  PROC DrawPart253()
    MoveL Offs(pOrigin,224.94,44.31,6.00),vTravel,z5,tPen\WObj:=wPaper;
    MoveL Offs(pOrigin,224.94,44.31,0.00),v60,z0,tPen\WObj:=wPaper;
    MoveL Offs(pOrigin,224.94,40.70,0.00),v40,z0,tPen\WObj:=wPaper;
    MoveL Offs(pOrigin,224.78,39.89,0.00),v40,z0,tPen\WObj:=wPaper;
    MoveL Offs(pOrigin,227.34,42.45,0.00),v40,z0,tPen\WObj:=wPaper;
    MoveL Offs(pOrigin,226.84,42.46,0.00),v40,z0,tPen\WObj:=wPaper;
    MoveL Offs(pOrigin,223.22,42.46,0.00),v40,fine,tPen\WObj:=wPaper;
    MoveL Offs(pOrigin,223.22,42.46,6.00),v60,z5,tPen\WObj:=wPaper;
    MoveL Offs(pOrigin,222.09,40.18,6.00),vTravel,z5,tPen\WObj:=wPaper;
    MoveL Offs(pOrigin,222.09,40.18,0.00),v60,z0,tPen\WObj:=wPaper;
    MoveL Offs(pOrigin,226.29,44.39,0.00),v40,z0,tPen\WObj:=wPaper;
    MoveL Offs(pOrigin,226.74,43.34,0.00),v40,z0,tPen\WObj:=wPaper;
    MoveL Offs(pOrigin,223.28,39.89,0.00),v40,z0,tPen\WObj:=wPaper;
    MoveL Offs(pOrigin,223.66,39.43,0.00),v40,z0,tPen\WObj:=wPaper;
    MoveL Offs(pOrigin,205.18,57.91,0.00),v40,z0,tPen\WObj:=wPaper;
    MoveL Offs(pOrigin,204.91,57.36,0.00),v40,z0,tPen\WObj:=wPaper;
    MoveL Offs(pOrigin,203.56,56.00,0.00),v40,z0,tPen\WObj:=wPaper;
    MoveL Offs(pOrigin,203.09,55.52,0.00),v40,z0,tPen\WObj:=wPaper;
    MoveL Offs(pOrigin,197.53,61.08,0.00),v40,z0,tPen\WObj:=wPaper;
    MoveL Offs(pOrigin,197.58,60.48,0.00),v40,z0,tPen\WObj:=wPaper;
    MoveL Offs(pOrigin,196.23,59.13,0.00),v40,z0,tPen\WObj:=wPaper;
    MoveL Offs(pOrigin,196.66,59.35,0.00),v40,z0,tPen\WObj:=wPaper;
    MoveL Offs(pOrigin,199.00,59.35,0.00),v40,z0,tPen\WObj:=wPaper;
    MoveL Offs(pOrigin,198.78,60.18,0.00),v40,z0,tPen\WObj:=wPaper;
    MoveL Offs(pOrigin,197.28,58.68,0.00),v40,z0,tPen\WObj:=wPaper;
    MoveL Offs(pOrigin,197.69,57.93,0.00),v40,z0,tPen\WObj:=wPaper;
    MoveL Offs(pOrigin,193.48,62.14,0.00),v40,z0,tPen\WObj:=wPaper;
    MoveL Offs(pOrigin,192.94,61.81,0.00),v40,z0,tPen\WObj:=wPaper;
    MoveL Offs(pOrigin,191.74,60.61,0.00),v40,z0,tPen\WObj:=wPaper;
    MoveL Offs(pOrigin,191.39,59.75,0.00),v40,z0,tPen\WObj:=wPaper;
    MoveL Offs(pOrigin,187.04,64.10,0.00),v40,z0,tPen\WObj:=wPaper;
    MoveL Offs(pOrigin,186.95,63.29,0.00),v40,z0,tPen\WObj:=wPaper;
    MoveL Offs(pOrigin,186.05,62.39,0.00),v40,z0,tPen\WObj:=wPaper;
    MoveL Offs(pOrigin,187.10,61.95,0.00),v40,z0,tPen\WObj:=wPaper;
    MoveL Offs(pOrigin,188.30,63.15,0.00),v40,z0,tPen\WObj:=wPaper;
    MoveL Offs(pOrigin,189.44,63.20,0.00),v40,z0,tPen\WObj:=wPaper;
    MoveL Offs(pOrigin,193.49,59.14,0.00),v40,z0,tPen\WObj:=wPaper;
    MoveL Offs(pOrigin,193.98,59.87,0.00),v40,z0,tPen\WObj:=wPaper;
    MoveL Offs(pOrigin,195.34,61.22,0.00),v40,z0,tPen\WObj:=wPaper;
    MoveL Offs(pOrigin,195.43,61.68,0.00),v40,z0,tPen\WObj:=wPaper;
    MoveL Offs(pOrigin,200.39,56.72,0.00),v40,z0,tPen\WObj:=wPaper;
    MoveL Offs(pOrigin,200.72,57.64,0.00),v40,z0,tPen\WObj:=wPaper;
    MoveL Offs(pOrigin,202.07,59.00,0.00),v40,z0,tPen\WObj:=wPaper;
    MoveL Offs(pOrigin,202.48,59.11,0.00),v40,z0,tPen\WObj:=wPaper;
    MoveL Offs(pOrigin,210.15,51.45,0.00),v40,z0,tPen\WObj:=wPaper;
    MoveL Offs(pOrigin,210.14,52.13,0.00),v40,z0,tPen\WObj:=wPaper;
    MoveL Offs(pOrigin,211.79,53.78,0.00),v40,z0,tPen\WObj:=wPaper;
    MoveL Offs(pOrigin,211.33,54.74,0.00),v40,z0,tPen\WObj:=wPaper;
    MoveL Offs(pOrigin,226.96,39.12,0.00),v40,z0,tPen\WObj:=wPaper;
    MoveL Offs(pOrigin,227.63,39.75,0.00),v40,z0,tPen\WObj:=wPaper;
    MoveL Offs(pOrigin,229.58,41.70,0.00),v40,fine,tPen\WObj:=wPaper;
    MoveL Offs(pOrigin,229.58,41.70,6.00),v60,z5,tPen\WObj:=wPaper;
    MoveL Offs(pOrigin,227.05,41.55,6.00),vTravel,z5,tPen\WObj:=wPaper;
    MoveL Offs(pOrigin,227.05,41.55,0.00),v60,z0,tPen\WObj:=wPaper;
    MoveL Offs(pOrigin,227.05,40.49,0.00),v40,fine,tPen\WObj:=wPaper;
    MoveL Offs(pOrigin,227.05,40.49,6.00),v60,z5,tPen\WObj:=wPaper;
    MoveL Offs(pOrigin,225.46,39.12,6.00),vTravel,z5,tPen\WObj:=wPaper;
    MoveL Offs(pOrigin,225.46,39.12,0.00),v60,z0,tPen\WObj:=wPaper;
    MoveL Offs(pOrigin,208.78,55.80,0.00),v40,z0,tPen\WObj:=wPaper;
    MoveL Offs(pOrigin,208.80,55.27,0.00),v40,z0,tPen\WObj:=wPaper;
    MoveL Offs(pOrigin,207.45,53.92,0.00),v40,z0,tPen\WObj:=wPaper;
    MoveL Offs(pOrigin,207.92,54.07,0.00),v40,z0,tPen\WObj:=wPaper;
    MoveL Offs(pOrigin,209.84,54.07,0.00),v40,z0,tPen\WObj:=wPaper;
    MoveL Offs(pOrigin,209.85,54.83,0.00),v40,z0,tPen\WObj:=wPaper;
    MoveL Offs(pOrigin,208.34,53.32,0.00),v40,z0,tPen\WObj:=wPaper;
    MoveL Offs(pOrigin,209.39,52.88,0.00),v40,z0,tPen\WObj:=wPaper;
    MoveL Offs(pOrigin,210.74,54.23,0.00),v40,fine,tPen\WObj:=wPaper;
    MoveL Offs(pOrigin,210.74,54.23,6.00),v60,z5,tPen\WObj:=wPaper;
    MoveL Offs(pOrigin,209.62,53.02,6.00),vTravel,z5,tPen\WObj:=wPaper;
    MoveL Offs(pOrigin,209.62,53.02,0.00),v60,z0,tPen\WObj:=wPaper;
    MoveL Offs(pOrigin,218.76,53.02,0.00),v40,z0,tPen\WObj:=wPaper;
    MoveL Offs(pOrigin,218.98,52.81,0.00),v40,z0,tPen\WObj:=wPaper;
    MoveL Offs(pOrigin,217.91,53.88,0.00),v40,z0,tPen\WObj:=wPaper;
    MoveL Offs(pOrigin,218.98,52.81,0.00),v40,z0,tPen\WObj:=wPaper;
    MoveL Offs(pOrigin,218.98,53.51,0.00),v40,z0,tPen\WObj:=wPaper;
    MoveL Offs(pOrigin,217.03,51.55,0.00),v40,fine,tPen\WObj:=wPaper;
    MoveL Offs(pOrigin,217.03,51.55,6.00),v60,z5,tPen\WObj:=wPaper;
    MoveL Offs(pOrigin,215.79,53.88,6.00),vTravel,z5,tPen\WObj:=wPaper;
    MoveL Offs(pOrigin,215.79,53.88,0.00),v60,z0,tPen\WObj:=wPaper;
    MoveL Offs(pOrigin,216.21,54.30,0.00),v40,z0,tPen\WObj:=wPaper;
    MoveL Offs(pOrigin,215.79,53.88,0.00),v40,fine,tPen\WObj:=wPaper;
    MoveL Offs(pOrigin,215.79,53.88,6.00),v60,z5,tPen\WObj:=wPaper;
    MoveL Offs(pOrigin,216.64,55.13,6.00),vTravel,z5,tPen\WObj:=wPaper;
    MoveL Offs(pOrigin,216.64,55.13,0.00),v60,z0,tPen\WObj:=wPaper;
    MoveL Offs(pOrigin,217.91,55.13,0.00),v40,z0,tPen\WObj:=wPaper;
    MoveL Offs(pOrigin,217.91,56.18,0.00),v40,z0,tPen\WObj:=wPaper;
    MoveL Offs(pOrigin,216.85,56.18,0.00),v40,fine,tPen\WObj:=wPaper;
    MoveL Offs(pOrigin,216.85,56.18,6.00),v60,z5,tPen\WObj:=wPaper;
    MoveL Offs(pOrigin,218.66,57.87,6.00),vTravel,z5,tPen\WObj:=wPaper;
    MoveL Offs(pOrigin,218.66,57.87,0.00),v60,z0,tPen\WObj:=wPaper;
    MoveL Offs(pOrigin,208.75,67.78,0.00),v40,z0,tPen\WObj:=wPaper;
    MoveL Offs(pOrigin,208.84,67.26,0.00),v40,z0,tPen\WObj:=wPaper;
    MoveL Offs(pOrigin,207.33,65.75,0.00),v40,z0,tPen\WObj:=wPaper;
    MoveL Offs(pOrigin,206.36,65.69,0.00),v40,z0,tPen\WObj:=wPaper;
    MoveL Offs(pOrigin,192.23,79.82,0.00),v40,z0,tPen\WObj:=wPaper;
    MoveL Offs(pOrigin,192.24,79.04,0.00),v40,z0,tPen\WObj:=wPaper;
    MoveL Offs(pOrigin,188.19,74.98,0.00),v40,z0,tPen\WObj:=wPaper;
    MoveL Offs(pOrigin,188.16,75.19,0.00),v40,z0,tPen\WObj:=wPaper;
    MoveL Offs(pOrigin,206.65,75.19,0.00),v40,z0,tPen\WObj:=wPaper;
    MoveL Offs(pOrigin,206.86,74.14,0.00),v40,z0,tPen\WObj:=wPaper;
    MoveL Offs(pOrigin,210.48,74.14,0.00),v40,z0,tPen\WObj:=wPaper;
    MoveL Offs(pOrigin,210.51,74.90,0.00),v40,z0,tPen\WObj:=wPaper;
    MoveL Offs(pOrigin,208.85,73.25,0.00),v40,z0,tPen\WObj:=wPaper;
    MoveL Offs(pOrigin,208.58,72.43,0.00),v40,z0,tPen\WObj:=wPaper;
    MoveL Offs(pOrigin,204.53,76.48,0.00),v40,z0,tPen\WObj:=wPaper;
    MoveL Offs(pOrigin,204.52,76.38,0.00),v40,z0,tPen\WObj:=wPaper;
    MoveL Offs(pOrigin,202.72,74.58,0.00),v40,z0,tPen\WObj:=wPaper;
    MoveL Offs(pOrigin,202.74,73.79,0.00),v40,z0,tPen\WObj:=wPaper;
    MoveL Offs(pOrigin,199.58,76.95,0.00),v40,z0,tPen\WObj:=wPaper;
    MoveL Offs(pOrigin,200.18,76.52,0.00),v40,z0,tPen\WObj:=wPaper;
    MoveL Offs(pOrigin,195.37,71.71,0.00),v40,z0,tPen\WObj:=wPaper;
    MoveL Offs(pOrigin,195.60,72.02,0.00),v40,z0,tPen\WObj:=wPaper;
    MoveL Offs(pOrigin,199.00,72.02,0.00),v40,z0,tPen\WObj:=wPaper;
    MoveL Offs(pOrigin,199.21,72.36,0.00),v40,z0,tPen\WObj:=wPaper;
    MoveL Offs(pOrigin,199.43,71.94,0.00),v40,z0,tPen\WObj:=wPaper;
    MoveL Offs(pOrigin,199.21,72.36,0.00),v40,z0,tPen\WObj:=wPaper;
    MoveL Offs(pOrigin,199.42,72.77,0.00),v40,z0,tPen\WObj:=wPaper;
    MoveL Offs(pOrigin,197.61,70.97,0.00),v40,z0,tPen\WObj:=wPaper;
    MoveL Offs(pOrigin,197.94,70.97,0.00),v40,z0,tPen\WObj:=wPaper;
    MoveL Offs(pOrigin,200.49,70.97,0.00),v40,z0,tPen\WObj:=wPaper;
  ENDPROC

  PROC DrawPart254()
    MoveL Offs(pOrigin,201.06,71.43,0.00),v40,z0,tPen\WObj:=wPaper;
    MoveL Offs(pOrigin,199.71,70.07,0.00),v40,z0,tPen\WObj:=wPaper;
    MoveL Offs(pOrigin,199.90,69.16,0.00),v40,z0,tPen\WObj:=wPaper;
    MoveL Offs(pOrigin,171.05,98.01,0.00),v40,z0,tPen\WObj:=wPaper;
    MoveL Offs(pOrigin,170.58,97.70,0.00),v40,z0,tPen\WObj:=wPaper;
    MoveL Offs(pOrigin,165.32,92.44,0.00),v40,z0,tPen\WObj:=wPaper;
    MoveL Offs(pOrigin,165.64,92.55,0.00),v40,z0,tPen\WObj:=wPaper;
    MoveL Offs(pOrigin,165.21,93.19,0.00),v40,z0,tPen\WObj:=wPaper;
    MoveL Offs(pOrigin,165.64,92.55,0.00),v40,z0,tPen\WObj:=wPaper;
    MoveL Offs(pOrigin,165.42,93.14,0.00),v40,z0,tPen\WObj:=wPaper;
    MoveL Offs(pOrigin,167.98,93.14,0.00),v40,z0,tPen\WObj:=wPaper;
    MoveL Offs(pOrigin,167.98,93.40,0.00),v40,z0,tPen\WObj:=wPaper;
    MoveL Offs(pOrigin,168.12,92.34,0.00),v40,z0,tPen\WObj:=wPaper;
    MoveL Offs(pOrigin,168.82,91.28,0.00),v40,z0,tPen\WObj:=wPaper;
    MoveL Offs(pOrigin,170.31,90.85,0.00),v40,z0,tPen\WObj:=wPaper;
    MoveL Offs(pOrigin,170.52,89.98,0.00),v40,z0,tPen\WObj:=wPaper;
    MoveL Offs(pOrigin,168.19,89.98,0.00),v40,z0,tPen\WObj:=wPaper;
    MoveL Offs(pOrigin,167.76,90.00,0.00),v40,z0,tPen\WObj:=wPaper;
    MoveL Offs(pOrigin,167.12,90.64,0.00),v40,z0,tPen\WObj:=wPaper;
    MoveL Offs(pOrigin,167.76,90.00,0.00),v40,z0,tPen\WObj:=wPaper;
    MoveL Offs(pOrigin,167.41,90.05,0.00),v40,z0,tPen\WObj:=wPaper;
    MoveL Offs(pOrigin,170.27,92.90,0.00),v40,z0,tPen\WObj:=wPaper;
    MoveL Offs(pOrigin,171.02,93.65,0.00),v40,z0,tPen\WObj:=wPaper;
    MoveL Offs(pOrigin,173.87,96.51,0.00),v40,z0,tPen\WObj:=wPaper;
    MoveL Offs(pOrigin,172.98,97.11,0.00),v40,z0,tPen\WObj:=wPaper;
    MoveL Offs(pOrigin,170.42,94.55,0.00),v40,z0,tPen\WObj:=wPaper;
    MoveL Offs(pOrigin,169.68,95.26,0.00),v40,z0,tPen\WObj:=wPaper;
    MoveL Offs(pOrigin,173.92,95.26,0.00),v40,z0,tPen\WObj:=wPaper;
    MoveL Offs(pOrigin,174.47,95.61,0.00),v40,z0,tPen\WObj:=wPaper;
    MoveL Offs(pOrigin,171.92,93.06,0.00),v40,z0,tPen\WObj:=wPaper;
    MoveL Offs(pOrigin,172.66,92.31,0.00),v40,z0,tPen\WObj:=wPaper;
    MoveL Offs(pOrigin,175.22,94.87,0.00),v40,z0,tPen\WObj:=wPaper;
    MoveL Offs(pOrigin,174.99,94.46,0.00),v40,z0,tPen\WObj:=wPaper;
    MoveL Offs(pOrigin,174.35,95.10,0.00),v40,z0,tPen\WObj:=wPaper;
    MoveL Offs(pOrigin,174.99,94.46,0.00),v40,z0,tPen\WObj:=wPaper;
    MoveL Offs(pOrigin,175.20,94.20,0.00),v40,z0,tPen\WObj:=wPaper;
    MoveL Offs(pOrigin,172.01,94.20,0.00),v40,fine,tPen\WObj:=wPaper;
    MoveL Offs(pOrigin,172.01,94.20,6.00),v60,z5,tPen\WObj:=wPaper;
    MoveL Offs(pOrigin,173.08,93.14,6.00),vTravel,z5,tPen\WObj:=wPaper;
    MoveL Offs(pOrigin,173.08,93.14,0.00),v60,z0,tPen\WObj:=wPaper;
    MoveL Offs(pOrigin,176.69,93.14,0.00),v40,z0,tPen\WObj:=wPaper;
    MoveL Offs(pOrigin,176.90,92.97,0.00),v40,z0,tPen\WObj:=wPaper;
    MoveL Offs(pOrigin,176.48,93.40,0.00),v40,z0,tPen\WObj:=wPaper;
    MoveL Offs(pOrigin,176.90,92.97,0.00),v40,z0,tPen\WObj:=wPaper;
    MoveL Offs(pOrigin,176.86,93.52,0.00),v40,z0,tPen\WObj:=wPaper;
    MoveL Offs(pOrigin,174.31,90.97,0.00),v40,z0,tPen\WObj:=wPaper;
    MoveL Offs(pOrigin,173.56,91.71,0.00),v40,z0,tPen\WObj:=wPaper;
    MoveL Offs(pOrigin,175.96,94.12,0.00),v40,z0,tPen\WObj:=wPaper;
    MoveL Offs(pOrigin,176.05,93.61,0.00),v40,z0,tPen\WObj:=wPaper;
    MoveL Offs(pOrigin,175.41,94.25,0.00),v40,z0,tPen\WObj:=wPaper;
    MoveL Offs(pOrigin,176.05,93.61,0.00),v40,fine,tPen\WObj:=wPaper;
    MoveL Offs(pOrigin,176.05,93.61,6.00),v60,z5,tPen\WObj:=wPaper;
    MoveL Offs(pOrigin,174.35,92.09,6.00),vTravel,z5,tPen\WObj:=wPaper;
    MoveL Offs(pOrigin,174.35,92.09,0.00),v60,z0,tPen\WObj:=wPaper;
    MoveL Offs(pOrigin,177.96,92.09,0.00),v40,z0,tPen\WObj:=wPaper;
    MoveL Offs(pOrigin,178.65,92.33,0.00),v40,z0,tPen\WObj:=wPaper;
    MoveL Offs(pOrigin,175.95,89.62,0.00),v40,z0,tPen\WObj:=wPaper;
    MoveL Offs(pOrigin,176.90,89.98,0.00),v40,z0,tPen\WObj:=wPaper;
    MoveL Offs(pOrigin,180.30,89.98,0.00),v40,z0,tPen\WObj:=wPaper;
    MoveL Offs(pOrigin,181.04,90.24,0.00),v40,z0,tPen\WObj:=wPaper;
    MoveL Offs(pOrigin,178.49,87.69,0.00),v40,z0,tPen\WObj:=wPaper;
    MoveL Offs(pOrigin,179.45,87.86,0.00),v40,z0,tPen\WObj:=wPaper;
    MoveL Offs(pOrigin,182.85,87.86,0.00),v40,z0,tPen\WObj:=wPaper;
    MoveL Offs(pOrigin,183.28,88.00,0.00),v40,z0,tPen\WObj:=wPaper;
    MoveL Offs(pOrigin,180.73,85.44,0.00),v40,z0,tPen\WObj:=wPaper;
    MoveL Offs(pOrigin,181.63,84.85,0.00),v40,z0,tPen\WObj:=wPaper;
    MoveL Offs(pOrigin,184.18,87.40,0.00),v40,z0,tPen\WObj:=wPaper;
    MoveL Offs(pOrigin,183.70,87.24,0.00),v40,z0,tPen\WObj:=wPaper;
    MoveL Offs(pOrigin,182.85,88.09,0.00),v40,z0,tPen\WObj:=wPaper;
    MoveL Offs(pOrigin,183.70,87.24,0.00),v40,z0,tPen\WObj:=wPaper;
    MoveL Offs(pOrigin,184.12,86.81,0.00),v40,z0,tPen\WObj:=wPaper;
    MoveL Offs(pOrigin,180.94,86.81,0.00),v40,z0,tPen\WObj:=wPaper;
    MoveL Offs(pOrigin,180.13,86.34,0.00),v40,z0,tPen\WObj:=wPaper;
    MoveL Offs(pOrigin,182.54,88.75,0.00),v40,z0,tPen\WObj:=wPaper;
    MoveL Offs(pOrigin,182.00,88.72,0.00),v40,z0,tPen\WObj:=wPaper;
    MoveL Offs(pOrigin,181.15,89.57,0.00),v40,z0,tPen\WObj:=wPaper;
    MoveL Offs(pOrigin,182.00,88.72,0.00),v40,z0,tPen\WObj:=wPaper;
    MoveL Offs(pOrigin,181.58,88.92,0.00),v40,z0,tPen\WObj:=wPaper;
    MoveL Offs(pOrigin,178.18,88.92,0.00),v40,fine,tPen\WObj:=wPaper;
    MoveL Offs(pOrigin,178.18,88.92,6.00),v60,z5,tPen\WObj:=wPaper;
    MoveL Offs(pOrigin,176.70,88.88,6.00),vTravel,z5,tPen\WObj:=wPaper;
    MoveL Offs(pOrigin,176.70,88.88,0.00),v60,z0,tPen\WObj:=wPaper;
    MoveL Offs(pOrigin,179.40,91.58,0.00),v40,fine,tPen\WObj:=wPaper;
    MoveL Offs(pOrigin,179.40,91.58,6.00),v60,z5,tPen\WObj:=wPaper;
    MoveL Offs(pOrigin,181.64,89.34,6.00),vTravel,z5,tPen\WObj:=wPaper;
    MoveL Offs(pOrigin,181.64,89.34,0.00),v60,z0,tPen\WObj:=wPaper;
    MoveL Offs(pOrigin,179.24,86.94,0.00),v40,fine,tPen\WObj:=wPaper;
    MoveL Offs(pOrigin,179.24,86.94,6.00),v60,z5,tPen\WObj:=wPaper;
    MoveL Offs(pOrigin,182.00,85.75,6.00),vTravel,z5,tPen\WObj:=wPaper;
    MoveL Offs(pOrigin,182.00,85.75,0.00),v60,z0,tPen\WObj:=wPaper;
    MoveL Offs(pOrigin,184.98,85.75,0.00),v40,z0,tPen\WObj:=wPaper;
    MoveL Offs(pOrigin,185.40,85.75,0.00),v40,z0,tPen\WObj:=wPaper;
    MoveL Offs(pOrigin,184.34,86.81,0.00),v40,z0,tPen\WObj:=wPaper;
    MoveL Offs(pOrigin,185.40,85.75,0.00),v40,z0,tPen\WObj:=wPaper;
    MoveL Offs(pOrigin,185.83,86.06,0.00),v40,z0,tPen\WObj:=wPaper;
    MoveL Offs(pOrigin,183.12,83.36,0.00),v40,z0,tPen\WObj:=wPaper;
    MoveL Offs(pOrigin,182.37,84.10,0.00),v40,z0,tPen\WObj:=wPaper;
    MoveL Offs(pOrigin,184.93,86.66,0.00),v40,fine,tPen\WObj:=wPaper;
    MoveL Offs(pOrigin,184.93,86.66,6.00),v60,z5,tPen\WObj:=wPaper;
    MoveL Offs(pOrigin,183.37,88.68,6.00),vTravel,z5,tPen\WObj:=wPaper;
    MoveL Offs(pOrigin,183.37,88.68,0.00),v60,z0,tPen\WObj:=wPaper;
    MoveL Offs(pOrigin,191.33,80.72,0.00),v40,z0,tPen\WObj:=wPaper;
    MoveL Offs(pOrigin,190.75,80.53,0.00),v40,z0,tPen\WObj:=wPaper;
    MoveL Offs(pOrigin,185.94,75.72,0.00),v40,z0,tPen\WObj:=wPaper;
    MoveL Offs(pOrigin,185.19,76.25,0.00),v40,z0,tPen\WObj:=wPaper;
    MoveL Offs(pOrigin,189.23,76.25,0.00),v40,fine,tPen\WObj:=wPaper;
    MoveL Offs(pOrigin,189.23,76.25,6.00),v60,z5,tPen\WObj:=wPaper;
    MoveL Offs(pOrigin,190.50,77.30,6.00),vTravel,z5,tPen\WObj:=wPaper;
    MoveL Offs(pOrigin,190.50,77.30,0.00),v60,z0,tPen\WObj:=wPaper;
    MoveL Offs(pOrigin,193.48,77.30,0.00),v40,z0,tPen\WObj:=wPaper;
    MoveL Offs(pOrigin,193.89,77.70,0.00),v40,z0,tPen\WObj:=wPaper;
    MoveL Offs(pOrigin,190.28,74.09,0.00),v40,z0,tPen\WObj:=wPaper;
    MoveL Offs(pOrigin,190.92,74.14,0.00),v40,z0,tPen\WObj:=wPaper;
    MoveL Offs(pOrigin,197.30,74.14,0.00),v40,z0,tPen\WObj:=wPaper;
    MoveL Offs(pOrigin,197.51,73.85,0.00),v40,z0,tPen\WObj:=wPaper;
    MoveL Offs(pOrigin,197.73,73.43,0.00),v40,z0,tPen\WObj:=wPaper;
    MoveL Offs(pOrigin,197.51,73.85,0.00),v40,z0,tPen\WObj:=wPaper;
    MoveL Offs(pOrigin,197.49,73.21,0.00),v40,z0,tPen\WObj:=wPaper;
    MoveL Offs(pOrigin,197.49,71.72,0.00),v40,z0,tPen\WObj:=wPaper;
    MoveL Offs(pOrigin,196.57,71.41,0.00),v40,z0,tPen\WObj:=wPaper;
  ENDPROC

  PROC DrawPart255()
    MoveL Offs(pOrigin,198.52,73.37,0.00),v40,z0,tPen\WObj:=wPaper;
    MoveL Offs(pOrigin,198.15,73.21,0.00),v40,z0,tPen\WObj:=wPaper;
    MoveL Offs(pOrigin,198.57,73.00,0.00),v40,z0,tPen\WObj:=wPaper;
    MoveL Offs(pOrigin,198.15,73.21,0.00),v40,z0,tPen\WObj:=wPaper;
    MoveL Offs(pOrigin,198.15,73.08,0.00),v40,z0,tPen\WObj:=wPaper;
    MoveL Offs(pOrigin,193.26,73.08,0.00),v40,z0,tPen\WObj:=wPaper;
    MoveL Offs(pOrigin,193.57,72.90,0.00),v40,z0,tPen\WObj:=wPaper;
    MoveL Offs(pOrigin,197.33,76.66,0.00),v40,z0,tPen\WObj:=wPaper;
    MoveL Offs(pOrigin,198.08,76.95,0.00),v40,z0,tPen\WObj:=wPaper;
    MoveL Offs(pOrigin,201.09,73.95,0.00),v40,z0,tPen\WObj:=wPaper;
    MoveL Offs(pOrigin,201.22,74.57,0.00),v40,z0,tPen\WObj:=wPaper;
    MoveL Offs(pOrigin,203.02,76.38,0.00),v40,z0,tPen\WObj:=wPaper;
    MoveL Offs(pOrigin,202.73,76.79,0.00),v40,z0,tPen\WObj:=wPaper;
    MoveL Offs(pOrigin,206.48,73.03,0.00),v40,z0,tPen\WObj:=wPaper;
    MoveL Offs(pOrigin,206.61,73.99,0.00),v40,z0,tPen\WObj:=wPaper;
    MoveL Offs(pOrigin,208.26,75.64,0.00),v40,fine,tPen\WObj:=wPaper;
    MoveL Offs(pOrigin,208.26,75.64,6.00),v60,z5,tPen\WObj:=wPaper;
    MoveL Offs(pOrigin,209.46,75.35,6.00),vTravel,z5,tPen\WObj:=wPaper;
    MoveL Offs(pOrigin,209.46,75.35,0.00),v60,z0,tPen\WObj:=wPaper;
    MoveL Offs(pOrigin,207.66,73.54,0.00),v40,fine,tPen\WObj:=wPaper;
    MoveL Offs(pOrigin,207.66,73.54,6.00),v60,z5,tPen\WObj:=wPaper;
    MoveL Offs(pOrigin,210.05,72.95,6.00),vTravel,z5,tPen\WObj:=wPaper;
    MoveL Offs(pOrigin,210.05,72.95,0.00),v60,z0,tPen\WObj:=wPaper;
    MoveL Offs(pOrigin,211.55,74.45,0.00),v40,fine,tPen\WObj:=wPaper;
    MoveL Offs(pOrigin,211.55,74.45,6.00),v60,z5,tPen\WObj:=wPaper;
    MoveL Offs(pOrigin,210.22,75.27,6.00),vTravel,z5,tPen\WObj:=wPaper;
    MoveL Offs(pOrigin,210.22,75.27,0.00),v60,z0,tPen\WObj:=wPaper;
    MoveL Offs(pOrigin,218.64,66.85,0.00),v40,fine,tPen\WObj:=wPaper;
    MoveL Offs(pOrigin,218.64,66.85,6.00),v60,z5,tPen\WObj:=wPaper;
    MoveL Offs(pOrigin,218.50,64.01,6.00),vTravel,z5,tPen\WObj:=wPaper;
    MoveL Offs(pOrigin,218.50,64.01,0.00),v60,z0,tPen\WObj:=wPaper;
    MoveL Offs(pOrigin,212.64,69.87,0.00),v40,z0,tPen\WObj:=wPaper;
    MoveL Offs(pOrigin,213.34,70.27,0.00),v40,z0,tPen\WObj:=wPaper;
    MoveL Offs(pOrigin,214.99,71.92,0.00),v40,z0,tPen\WObj:=wPaper;
    MoveL Offs(pOrigin,214.94,71.09,0.00),v40,z0,tPen\WObj:=wPaper;
    MoveL Offs(pOrigin,214.73,71.51,0.00),v40,z0,tPen\WObj:=wPaper;
    MoveL Offs(pOrigin,214.94,71.09,0.00),v40,z0,tPen\WObj:=wPaper;
    MoveL Offs(pOrigin,214.94,70.97,0.00),v40,z0,tPen\WObj:=wPaper;
    MoveL Offs(pOrigin,213.45,70.97,0.00),v40,z0,tPen\WObj:=wPaper;
    MoveL Offs(pOrigin,213.88,70.03,0.00),v40,z0,tPen\WObj:=wPaper;
    MoveL Offs(pOrigin,213.66,70.45,0.00),v40,z0,tPen\WObj:=wPaper;
    MoveL Offs(pOrigin,213.88,70.03,0.00),v40,fine,tPen\WObj:=wPaper;
    MoveL Offs(pOrigin,213.88,70.03,6.00),v60,z5,tPen\WObj:=wPaper;
    MoveL Offs(pOrigin,214.09,72.02,6.00),vTravel,z5,tPen\WObj:=wPaper;
    MoveL Offs(pOrigin,214.09,72.02,0.00),v60,z0,tPen\WObj:=wPaper;
    MoveL Offs(pOrigin,212.18,72.02,0.00),v40,z0,tPen\WObj:=wPaper;
    MoveL Offs(pOrigin,211.96,72.15,0.00),v40,z0,tPen\WObj:=wPaper;
    MoveL Offs(pOrigin,212.46,71.80,0.00),v40,z0,tPen\WObj:=wPaper;
    MoveL Offs(pOrigin,210.26,73.07,0.00),v40,z0,tPen\WObj:=wPaper;
    MoveL Offs(pOrigin,205.16,74.49,0.00),v40,z0,tPen\WObj:=wPaper;
    MoveL Offs(pOrigin,200.70,74.91,0.00),v40,z0,tPen\WObj:=wPaper;
    MoveL Offs(pOrigin,196.95,74.84,0.00),v40,z0,tPen\WObj:=wPaper;
    MoveL Offs(pOrigin,197.37,73.85,0.00),v40,z0,tPen\WObj:=wPaper;
    MoveL Offs(pOrigin,200.06,71.44,0.00),v40,z0,tPen\WObj:=wPaper;
    MoveL Offs(pOrigin,204.74,69.60,0.00),v40,z0,tPen\WObj:=wPaper;
    MoveL Offs(pOrigin,205.80,69.60,0.00),v40,z0,tPen\WObj:=wPaper;
    MoveL Offs(pOrigin,206.30,69.20,0.00),v40,z0,tPen\WObj:=wPaper;
    MoveL Offs(pOrigin,204.79,67.69,0.00),v40,z0,tPen\WObj:=wPaper;
    MoveL Offs(pOrigin,205.38,67.80,0.00),v40,z0,tPen\WObj:=wPaper;
    MoveL Offs(pOrigin,206.86,67.80,0.00),v40,z0,tPen\WObj:=wPaper;
    MoveL Offs(pOrigin,207.07,67.90,0.00),v40,z0,tPen\WObj:=wPaper;
    MoveL Offs(pOrigin,206.65,68.32,0.00),v40,z0,tPen\WObj:=wPaper;
    MoveL Offs(pOrigin,207.07,67.90,0.00),v40,z0,tPen\WObj:=wPaper;
    MoveL Offs(pOrigin,207.04,68.45,0.00),v40,z0,tPen\WObj:=wPaper;
    MoveL Offs(pOrigin,205.69,67.10,0.00),v40,z0,tPen\WObj:=wPaper;
    MoveL Offs(pOrigin,206.59,66.50,0.00),v40,z0,tPen\WObj:=wPaper;
    MoveL Offs(pOrigin,207.94,67.85,0.00),v40,z0,tPen\WObj:=wPaper;
    MoveL Offs(pOrigin,208.14,67.05,0.00),v40,z0,tPen\WObj:=wPaper;
    MoveL Offs(pOrigin,207.50,67.69,0.00),v40,z0,tPen\WObj:=wPaper;
    MoveL Offs(pOrigin,208.14,67.05,0.00),v40,z0,tPen\WObj:=wPaper;
    MoveL Offs(pOrigin,208.14,66.74,0.00),v40,z0,tPen\WObj:=wPaper;
    MoveL Offs(pOrigin,206.86,66.74,0.00),v40,fine,tPen\WObj:=wPaper;
    MoveL Offs(pOrigin,206.86,66.74,6.00),v60,z5,tPen\WObj:=wPaper;
    MoveL Offs(pOrigin,208.35,65.69,6.00),vTravel,z5,tPen\WObj:=wPaper;
    MoveL Offs(pOrigin,208.35,65.69,0.00),v60,z0,tPen\WObj:=wPaper;
    MoveL Offs(pOrigin,209.62,65.69,0.00),v40,z0,tPen\WObj:=wPaper;
    MoveL Offs(pOrigin,209.84,65.78,0.00),v40,z0,tPen\WObj:=wPaper;
    MoveL Offs(pOrigin,209.41,66.20,0.00),v40,z0,tPen\WObj:=wPaper;
    MoveL Offs(pOrigin,209.84,65.78,0.00),v40,z0,tPen\WObj:=wPaper;
    MoveL Offs(pOrigin,210.33,65.76,0.00),v40,z0,tPen\WObj:=wPaper;
    MoveL Offs(pOrigin,208.98,64.41,0.00),v40,z0,tPen\WObj:=wPaper;
    MoveL Offs(pOrigin,209.62,64.63,0.00),v40,z0,tPen\WObj:=wPaper;
    MoveL Offs(pOrigin,210.90,64.63,0.00),v40,z0,tPen\WObj:=wPaper;
    MoveL Offs(pOrigin,210.90,64.93,0.00),v40,z0,tPen\WObj:=wPaper;
    MoveL Offs(pOrigin,210.48,65.35,0.00),v40,z0,tPen\WObj:=wPaper;
    MoveL Offs(pOrigin,210.90,64.93,0.00),v40,z0,tPen\WObj:=wPaper;
    MoveL Offs(pOrigin,211.23,65.17,0.00),v40,z0,tPen\WObj:=wPaper;
    MoveL Offs(pOrigin,209.87,63.81,0.00),v40,fine,tPen\WObj:=wPaper;
    MoveL Offs(pOrigin,209.87,63.81,6.00),v60,z5,tPen\WObj:=wPaper;
    MoveL Offs(pOrigin,211.75,64.29,6.00),vTravel,z5,tPen\WObj:=wPaper;
    MoveL Offs(pOrigin,211.75,64.29,0.00),v60,z0,tPen\WObj:=wPaper;
    MoveL Offs(pOrigin,211.32,64.71,0.00),v40,z0,tPen\WObj:=wPaper;
    MoveL Offs(pOrigin,211.75,64.29,0.00),v40,fine,tPen\WObj:=wPaper;
    MoveL Offs(pOrigin,211.75,64.29,6.00),v60,z5,tPen\WObj:=wPaper;
    MoveL Offs(pOrigin,213.66,62.80,6.00),vTravel,z5,tPen\WObj:=wPaper;
    MoveL Offs(pOrigin,213.66,62.80,0.00),v60,z0,tPen\WObj:=wPaper;
    MoveL Offs(pOrigin,213.24,63.22,0.00),v40,z0,tPen\WObj:=wPaper;
    MoveL Offs(pOrigin,213.66,62.80,0.00),v40,fine,tPen\WObj:=wPaper;
    MoveL Offs(pOrigin,213.66,62.80,6.00),v60,z5,tPen\WObj:=wPaper;
    MoveL Offs(pOrigin,212.60,61.95,6.00),vTravel,z5,tPen\WObj:=wPaper;
    MoveL Offs(pOrigin,212.60,61.95,0.00),v60,z0,tPen\WObj:=wPaper;
    MoveL Offs(pOrigin,211.96,62.59,0.00),v40,z0,tPen\WObj:=wPaper;
    MoveL Offs(pOrigin,212.60,61.95,0.00),v40,fine,tPen\WObj:=wPaper;
    MoveL Offs(pOrigin,212.60,61.95,6.00),v60,z5,tPen\WObj:=wPaper;
    MoveL Offs(pOrigin,213.40,66.12,6.00),vTravel,z5,tPen\WObj:=wPaper;
    MoveL Offs(pOrigin,213.40,66.12,0.00),v60,z0,tPen\WObj:=wPaper;
    MoveL Offs(pOrigin,218.20,61.31,0.00),v40,fine,tPen\WObj:=wPaper;
    MoveL Offs(pOrigin,218.20,61.31,6.00),v60,z5,tPen\WObj:=wPaper;
    MoveL Offs(pOrigin,218.20,62.81,6.00),vTravel,z5,tPen\WObj:=wPaper;
    MoveL Offs(pOrigin,218.20,62.81,0.00),v60,z0,tPen\WObj:=wPaper;
    MoveL Offs(pOrigin,213.39,67.62,0.00),v40,fine,tPen\WObj:=wPaper;
    MoveL Offs(pOrigin,213.39,67.62,6.00),v60,z5,tPen\WObj:=wPaper;
    MoveL Offs(pOrigin,209.73,66.66,6.00),vTravel,z5,tPen\WObj:=wPaper;
    MoveL Offs(pOrigin,209.73,66.66,0.00),v60,z0,tPen\WObj:=wPaper;
    MoveL Offs(pOrigin,208.23,65.16,0.00),v40,fine,tPen\WObj:=wPaper;
    MoveL Offs(pOrigin,208.23,65.16,6.00),v60,z5,tPen\WObj:=wPaper;
    MoveL Offs(pOrigin,205.59,68.86,6.00),vTravel,z5,tPen\WObj:=wPaper;
    MoveL Offs(pOrigin,205.59,68.86,0.00),v60,z0,tPen\WObj:=wPaper;
    MoveL Offs(pOrigin,203.46,68.86,0.00),v40,fine,tPen\WObj:=wPaper;
    MoveL Offs(pOrigin,203.46,68.86,6.00),v60,z5,tPen\WObj:=wPaper;
  ENDPROC

  PROC DrawPart256()
    MoveL Offs(pOrigin,200.01,71.87,6.00),vTravel,z5,tPen\WObj:=wPaper;
    MoveL Offs(pOrigin,200.01,71.87,0.00),v60,z0,tPen\WObj:=wPaper;
    MoveL Offs(pOrigin,198.66,70.52,0.00),v40,fine,tPen\WObj:=wPaper;
    MoveL Offs(pOrigin,198.66,70.52,6.00),v60,z5,tPen\WObj:=wPaper;
    MoveL Offs(pOrigin,197.35,70.21,6.00),vTravel,z5,tPen\WObj:=wPaper;
    MoveL Offs(pOrigin,197.35,70.21,0.00),v60,z0,tPen\WObj:=wPaper;
    MoveL Offs(pOrigin,169.11,98.46,0.00),v40,z0,tPen\WObj:=wPaper;
    MoveL Offs(pOrigin,169.38,97.99,0.00),v40,z0,tPen\WObj:=wPaper;
    MoveL Offs(pOrigin,160.07,88.68,0.00),v40,z0,tPen\WObj:=wPaper;
    MoveL Offs(pOrigin,160.54,88.92,0.00),v40,z0,tPen\WObj:=wPaper;
    MoveL Offs(pOrigin,161.81,88.92,0.00),v40,z0,tPen\WObj:=wPaper;
    MoveL Offs(pOrigin,161.81,87.86,0.00),v40,z0,tPen\WObj:=wPaper;
    MoveL Offs(pOrigin,160.54,87.86,0.00),v40,z0,tPen\WObj:=wPaper;
    MoveL Offs(pOrigin,160.54,86.81,0.00),v40,z0,tPen\WObj:=wPaper;
    MoveL Offs(pOrigin,161.60,86.81,0.00),v40,fine,tPen\WObj:=wPaper;
    MoveL Offs(pOrigin,161.60,86.81,6.00),v60,z5,tPen\WObj:=wPaper;
    MoveL Offs(pOrigin,161.39,84.70,6.00),vTravel,z5,tPen\WObj:=wPaper;
    MoveL Offs(pOrigin,161.39,84.70,0.00),v60,z0,tPen\WObj:=wPaper;
    MoveL Offs(pOrigin,160.11,84.70,0.00),v40,z0,tPen\WObj:=wPaper;
    MoveL Offs(pOrigin,159.11,84.56,0.00),v40,z0,tPen\WObj:=wPaper;
    MoveL Offs(pOrigin,161.97,81.71,0.00),v40,z0,tPen\WObj:=wPaper;
    MoveL Offs(pOrigin,161.52,80.66,0.00),v40,z0,tPen\WObj:=wPaper;
    MoveL Offs(pOrigin,158.97,83.22,0.00),v40,fine,tPen\WObj:=wPaper;
    MoveL Offs(pOrigin,158.97,83.22,6.00),v60,z5,tPen\WObj:=wPaper;
    MoveL Offs(pOrigin,160.11,83.64,6.00),vTravel,z5,tPen\WObj:=wPaper;
    MoveL Offs(pOrigin,160.11,83.64,0.00),v60,z0,tPen\WObj:=wPaper;
    MoveL Offs(pOrigin,161.18,83.64,0.00),v40,z0,tPen\WObj:=wPaper;
    MoveL Offs(pOrigin,162.11,83.06,0.00),v40,z0,tPen\WObj:=wPaper;
    MoveL Offs(pOrigin,159.11,86.06,0.00),v40,fine,tPen\WObj:=wPaper;
    MoveL Offs(pOrigin,159.11,86.06,6.00),v60,z5,tPen\WObj:=wPaper;
    MoveL Offs(pOrigin,159.25,88.91,6.00),vTravel,z5,tPen\WObj:=wPaper;
    MoveL Offs(pOrigin,159.25,88.91,0.00),v60,z0,tPen\WObj:=wPaper;
    MoveL Offs(pOrigin,167.81,80.34,0.00),v40,z0,tPen\WObj:=wPaper;
    MoveL Offs(pOrigin,167.53,79.71,0.00),v40,z0,tPen\WObj:=wPaper;
    MoveL Offs(pOrigin,166.33,78.51,0.00),v40,z0,tPen\WObj:=wPaper;
    MoveL Offs(pOrigin,165.87,77.80,0.00),v40,z0,tPen\WObj:=wPaper;
    MoveL Offs(pOrigin,172.79,70.89,0.00),v40,z0,tPen\WObj:=wPaper;
    MoveL Offs(pOrigin,171.89,70.29,0.00),v40,z0,tPen\WObj:=wPaper;
    MoveL Offs(pOrigin,165.88,76.30,0.00),v40,z0,tPen\WObj:=wPaper;
    MoveL Offs(pOrigin,165.27,75.96,0.00),v40,z0,tPen\WObj:=wPaper;
    MoveL Offs(pOrigin,156.26,66.94,0.00),v40,z0,tPen\WObj:=wPaper;
    MoveL Offs(pOrigin,156.47,66.30,0.00),v40,z0,tPen\WObj:=wPaper;
    MoveL Offs(pOrigin,151.51,71.25,0.00),v40,z0,tPen\WObj:=wPaper;
    MoveL Offs(pOrigin,151.17,70.82,0.00),v40,z0,tPen\WObj:=wPaper;
    MoveL Offs(pOrigin,135.70,55.35,0.00),v40,z0,tPen\WObj:=wPaper;
    MoveL Offs(pOrigin,136.31,55.13,0.00),v40,z0,tPen\WObj:=wPaper;
    MoveL Offs(pOrigin,137.38,55.13,0.00),v40,z0,tPen\WObj:=wPaper;
    MoveL Offs(pOrigin,137.38,54.07,0.00),v40,z0,tPen\WObj:=wPaper;
    MoveL Offs(pOrigin,136.10,54.07,0.00),v40,z0,tPen\WObj:=wPaper;
    MoveL Offs(pOrigin,136.10,53.02,0.00),v40,z0,tPen\WObj:=wPaper;
    MoveL Offs(pOrigin,143.75,53.02,0.00),v40,z0,tPen\WObj:=wPaper;
    MoveL Offs(pOrigin,143.54,51.96,0.00),v40,z0,tPen\WObj:=wPaper;
    MoveL Offs(pOrigin,136.10,51.96,0.00),v40,z0,tPen\WObj:=wPaper;
    MoveL Offs(pOrigin,135.54,52.20,0.00),v40,z0,tPen\WObj:=wPaper;
    MoveL Offs(pOrigin,155.67,72.34,0.00),v40,fine,tPen\WObj:=wPaper;
    MoveL Offs(pOrigin,155.67,72.34,6.00),v60,z5,tPen\WObj:=wPaper;
    MoveL Offs(pOrigin,155.25,71.09,6.00),vTravel,z5,tPen\WObj:=wPaper;
    MoveL Offs(pOrigin,155.25,71.09,0.00),v60,z0,tPen\WObj:=wPaper;
    MoveL Offs(pOrigin,155.25,67.69,0.00),v40,z0,tPen\WObj:=wPaper;
    MoveL Offs(pOrigin,155.01,66.74,0.00),v40,z0,tPen\WObj:=wPaper;
    MoveL Offs(pOrigin,145.45,66.74,0.00),v40,z0,tPen\WObj:=wPaper;
    MoveL Offs(pOrigin,145.74,66.62,0.00),v40,z0,tPen\WObj:=wPaper;
    MoveL Offs(pOrigin,145.74,63.86,0.00),v40,fine,tPen\WObj:=wPaper;
    MoveL Offs(pOrigin,145.74,63.86,6.00),v60,z5,tPen\WObj:=wPaper;
    MoveL Offs(pOrigin,146.80,64.92,6.00),vTravel,z5,tPen\WObj:=wPaper;
    MoveL Offs(pOrigin,146.80,64.92,0.00),v60,z0,tPen\WObj:=wPaper;
    MoveL Offs(pOrigin,146.80,67.47,0.00),v40,z0,tPen\WObj:=wPaper;
    MoveL Offs(pOrigin,147.15,67.80,0.00),v40,z0,tPen\WObj:=wPaper;
    MoveL Offs(pOrigin,158.41,67.80,0.00),v40,z0,tPen\WObj:=wPaper;
    MoveL Offs(pOrigin,158.36,67.55,0.00),v40,z0,tPen\WObj:=wPaper;
    MoveL Offs(pOrigin,166.47,75.66,0.00),v40,z0,tPen\WObj:=wPaper;
    MoveL Offs(pOrigin,166.27,75.34,0.00),v40,z0,tPen\WObj:=wPaper;
    MoveL Offs(pOrigin,166.70,75.12,0.00),v40,z0,tPen\WObj:=wPaper;
    MoveL Offs(pOrigin,166.27,75.34,0.00),v40,z0,tPen\WObj:=wPaper;
    MoveL Offs(pOrigin,165.42,75.19,0.00),v40,z0,tPen\WObj:=wPaper;
    MoveL Offs(pOrigin,160.75,75.19,0.00),v40,fine,tPen\WObj:=wPaper;
    MoveL Offs(pOrigin,160.75,75.19,6.00),v60,z5,tPen\WObj:=wPaper;
    MoveL Offs(pOrigin,162.24,76.25,6.00),vTravel,z5,tPen\WObj:=wPaper;
    MoveL Offs(pOrigin,162.24,76.25,0.00),v60,z0,tPen\WObj:=wPaper;
    MoveL Offs(pOrigin,158.20,76.25,0.00),v40,z0,tPen\WObj:=wPaper;
    MoveL Offs(pOrigin,158.41,76.82,0.00),v40,z0,tPen\WObj:=wPaper;
    MoveL Offs(pOrigin,158.41,78.31,0.00),v40,z0,tPen\WObj:=wPaper;
    MoveL Offs(pOrigin,158.20,78.36,0.00),v40,z0,tPen\WObj:=wPaper;
    MoveL Offs(pOrigin,159.90,78.36,0.00),v40,fine,tPen\WObj:=wPaper;
    MoveL Offs(pOrigin,159.90,78.36,6.00),v60,z5,tPen\WObj:=wPaper;
    MoveL Offs(pOrigin,160.93,77.59,6.00),vTravel,z5,tPen\WObj:=wPaper;
    MoveL Offs(pOrigin,160.93,77.59,0.00),v60,z0,tPen\WObj:=wPaper;
    MoveL Offs(pOrigin,156.88,73.54,0.00),v40,z0,tPen\WObj:=wPaper;
    MoveL Offs(pOrigin,157.32,72.49,0.00),v40,z0,tPen\WObj:=wPaper;
    MoveL Offs(pOrigin,135.68,50.85,0.00),v40,z0,tPen\WObj:=wPaper;
    MoveL Offs(pOrigin,136.10,50.90,0.00),v40,z0,tPen\WObj:=wPaper;
    MoveL Offs(pOrigin,143.32,50.90,0.00),v40,z0,tPen\WObj:=wPaper;
    MoveL Offs(pOrigin,144.09,50.30,0.00),v40,z0,tPen\WObj:=wPaper;
    MoveL Offs(pOrigin,136.12,58.27,0.00),v40,z0,tPen\WObj:=wPaper;
    MoveL Offs(pOrigin,136.95,57.91,0.00),v40,z0,tPen\WObj:=wPaper;
    MoveL Offs(pOrigin,137.16,58.34,0.00),v40,z0,tPen\WObj:=wPaper;
    MoveL Offs(pOrigin,136.95,57.91,0.00),v40,z0,tPen\WObj:=wPaper;
    MoveL Offs(pOrigin,137.38,58.30,0.00),v40,z0,tPen\WObj:=wPaper;
    MoveL Offs(pOrigin,138.65,58.30,0.00),v40,z0,tPen\WObj:=wPaper;
    MoveL Offs(pOrigin,138.65,57.91,0.00),v40,z0,tPen\WObj:=wPaper;
    MoveL Offs(pOrigin,138.86,58.34,0.00),v40,z0,tPen\WObj:=wPaper;
    MoveL Offs(pOrigin,138.65,57.91,0.00),v40,z0,tPen\WObj:=wPaper;
    MoveL Offs(pOrigin,138.01,57.24,0.00),v40,z0,tPen\WObj:=wPaper;
    MoveL Offs(pOrigin,136.95,57.24,0.00),v40,z0,tPen\WObj:=wPaper;
    MoveL Offs(pOrigin,136.15,57.30,0.00),v40,z0,tPen\WObj:=wPaper;
    MoveL Offs(pOrigin,148.17,69.32,0.00),v40,z0,tPen\WObj:=wPaper;
    MoveL Offs(pOrigin,148.37,69.92,0.00),v40,z0,tPen\WObj:=wPaper;
    MoveL Offs(pOrigin,153.48,64.81,0.00),v40,z0,tPen\WObj:=wPaper;
    MoveL Offs(pOrigin,153.26,65.44,0.00),v40,z0,tPen\WObj:=wPaper;
    MoveL Offs(pOrigin,164.22,76.41,0.00),v40,z0,tPen\WObj:=wPaper;
    MoveL Offs(pOrigin,163.93,76.76,0.00),v40,z0,tPen\WObj:=wPaper;
    MoveL Offs(pOrigin,171.14,69.55,0.00),v40,z0,tPen\WObj:=wPaper;
    MoveL Offs(pOrigin,170.25,68.95,0.00),v40,z0,tPen\WObj:=wPaper;
    MoveL Offs(pOrigin,161.68,77.51,0.00),v40,z0,tPen\WObj:=wPaper;
    MoveL Offs(pOrigin,161.98,77.15,0.00),v40,z0,tPen\WObj:=wPaper;
    MoveL Offs(pOrigin,158.07,73.24,0.00),v40,fine,tPen\WObj:=wPaper;
    MoveL Offs(pOrigin,158.07,73.24,6.00),v60,z5,tPen\WObj:=wPaper;
    MoveL Offs(pOrigin,158.41,71.30,6.00),vTravel,z5,tPen\WObj:=wPaper;
    MoveL Offs(pOrigin,158.41,71.30,0.00),v60,z0,tPen\WObj:=wPaper;
    MoveL Offs(pOrigin,158.41,68.32,0.00),v40,z0,tPen\WObj:=wPaper;
  ENDPROC

  PROC DrawPart257()
    MoveL Offs(pOrigin,157.36,68.11,0.00),v40,z0,tPen\WObj:=wPaper;
    MoveL Offs(pOrigin,157.36,71.30,0.00),v40,z0,tPen\WObj:=wPaper;
    MoveL Offs(pOrigin,156.30,71.09,0.00),v40,z0,tPen\WObj:=wPaper;
    MoveL Offs(pOrigin,156.30,67.90,0.00),v40,fine,tPen\WObj:=wPaper;
    MoveL Offs(pOrigin,156.30,67.90,6.00),v60,z5,tPen\WObj:=wPaper;
    MoveL Offs(pOrigin,156.07,69.39,6.00),vTravel,z5,tPen\WObj:=wPaper;
    MoveL Offs(pOrigin,156.07,69.39,0.00),v60,z0,tPen\WObj:=wPaper;
    MoveL Offs(pOrigin,156.93,70.24,0.00),v40,z0,tPen\WObj:=wPaper;
    MoveL Offs(pOrigin,159.90,70.24,0.00),v40,z0,tPen\WObj:=wPaper;
    MoveL Offs(pOrigin,161.81,69.81,0.00),v40,z0,tPen\WObj:=wPaper;
    MoveL Offs(pOrigin,161.58,70.88,0.00),v40,z0,tPen\WObj:=wPaper;
    MoveL Offs(pOrigin,161.58,68.54,0.00),v40,z0,tPen\WObj:=wPaper;
    MoveL Offs(pOrigin,160.53,68.54,0.00),v40,z0,tPen\WObj:=wPaper;
    MoveL Offs(pOrigin,160.53,71.09,0.00),v40,z0,tPen\WObj:=wPaper;
    MoveL Offs(pOrigin,159.47,71.09,0.00),v40,z0,tPen\WObj:=wPaper;
    MoveL Offs(pOrigin,159.47,68.54,0.00),v40,fine,tPen\WObj:=wPaper;
    MoveL Offs(pOrigin,159.47,68.54,6.00),v60,z5,tPen\WObj:=wPaper;
    MoveL Offs(pOrigin,158.87,66.89,6.00),vTravel,z5,tPen\WObj:=wPaper;
    MoveL Offs(pOrigin,158.87,66.89,0.00),v60,z0,tPen\WObj:=wPaper;
    MoveL Offs(pOrigin,150.30,75.45,0.00),v40,fine,tPen\WObj:=wPaper;
    MoveL Offs(pOrigin,150.30,75.45,6.00),v60,z5,tPen\WObj:=wPaper;
    MoveL Offs(pOrigin,151.19,77.55,6.00),vTravel,z5,tPen\WObj:=wPaper;
    MoveL Offs(pOrigin,151.19,77.55,0.00),v60,z0,tPen\WObj:=wPaper;
    MoveL Offs(pOrigin,142.78,85.96,0.00),v40,z0,tPen\WObj:=wPaper;
    MoveL Offs(pOrigin,142.23,85.78,0.00),v40,z0,tPen\WObj:=wPaper;
    MoveL Offs(pOrigin,138.63,82.17,0.00),v40,z0,tPen\WObj:=wPaper;
    MoveL Offs(pOrigin,138.15,81.63,0.00),v40,z0,tPen\WObj:=wPaper;
    MoveL Offs(pOrigin,134.69,85.09,0.00),v40,z0,tPen\WObj:=wPaper;
    MoveL Offs(pOrigin,134.74,84.26,0.00),v40,z0,tPen\WObj:=wPaper;
    MoveL Offs(pOrigin,133.09,82.60,0.00),v40,z0,tPen\WObj:=wPaper;
    MoveL Offs(pOrigin,133.20,82.10,0.00),v40,z0,tPen\WObj:=wPaper;
    MoveL Offs(pOrigin,130.35,84.95,0.00),v40,z0,tPen\WObj:=wPaper;
    MoveL Offs(pOrigin,130.69,84.69,0.00),v40,z0,tPen\WObj:=wPaper;
    MoveL Offs(pOrigin,127.99,81.99,0.00),v40,z0,tPen\WObj:=wPaper;
    MoveL Offs(pOrigin,128.11,81.21,0.00),v40,z0,tPen\WObj:=wPaper;
    MoveL Offs(pOrigin,124.81,84.52,0.00),v40,z0,tPen\WObj:=wPaper;
    MoveL Offs(pOrigin,124.10,84.07,0.00),v40,z0,tPen\WObj:=wPaper;
    MoveL Offs(pOrigin,121.70,81.67,0.00),v40,fine,tPen\WObj:=wPaper;
    MoveL Offs(pOrigin,121.70,81.67,6.00),v60,z5,tPen\WObj:=wPaper;
    MoveL Offs(pOrigin,121.22,83.63,6.00),vTravel,z5,tPen\WObj:=wPaper;
    MoveL Offs(pOrigin,121.22,83.63,0.00),v60,z0,tPen\WObj:=wPaper;
    MoveL Offs(pOrigin,124.67,80.17,0.00),v40,z0,tPen\WObj:=wPaper;
    MoveL Offs(pOrigin,123.62,79.73,0.00),v40,z0,tPen\WObj:=wPaper;
    MoveL Offs(pOrigin,120.17,83.18,0.00),v40,z0,tPen\WObj:=wPaper;
    MoveL Offs(pOrigin,119.12,82.74,0.00),v40,z0,tPen\WObj:=wPaper;
    MoveL Offs(pOrigin,122.73,79.13,0.00),v40,z0,tPen\WObj:=wPaper;
    MoveL Offs(pOrigin,121.68,78.69,0.00),v40,z0,tPen\WObj:=wPaper;
    MoveL Offs(pOrigin,117.92,82.44,0.00),v40,z0,tPen\WObj:=wPaper;
    MoveL Offs(pOrigin,117.20,81.65,0.00),v40,z0,tPen\WObj:=wPaper;
    MoveL Offs(pOrigin,113.30,77.75,0.00),v40,z0,tPen\WObj:=wPaper;
    MoveL Offs(pOrigin,114.04,77.36,0.00),v40,z0,tPen\WObj:=wPaper;
    MoveL Offs(pOrigin,112.54,78.86,0.00),v40,z0,tPen\WObj:=wPaper;
    MoveL Offs(pOrigin,113.15,79.10,0.00),v40,z0,tPen\WObj:=wPaper;
    MoveL Offs(pOrigin,112.10,78.04,0.00),v40,z0,tPen\WObj:=wPaper;
    MoveL Offs(pOrigin,111.80,78.12,0.00),v40,z0,tPen\WObj:=wPaper;
    MoveL Offs(pOrigin,113.30,76.61,0.00),v40,z0,tPen\WObj:=wPaper;
    MoveL Offs(pOrigin,112.40,76.02,0.00),v40,z0,tPen\WObj:=wPaper;
    MoveL Offs(pOrigin,111.05,77.37,0.00),v40,z0,tPen\WObj:=wPaper;
    MoveL Offs(pOrigin,110.30,76.62,0.00),v40,z0,tPen\WObj:=wPaper;
    MoveL Offs(pOrigin,111.65,75.27,0.00),v40,z0,tPen\WObj:=wPaper;
    MoveL Offs(pOrigin,110.60,75.34,0.00),v40,z0,tPen\WObj:=wPaper;
    MoveL Offs(pOrigin,111.24,75.97,0.00),v40,z0,tPen\WObj:=wPaper;
    MoveL Offs(pOrigin,110.60,75.34,0.00),v40,z0,tPen\WObj:=wPaper;
    MoveL Offs(pOrigin,110.29,74.74,0.00),v40,z0,tPen\WObj:=wPaper;
    MoveL Offs(pOrigin,107.89,72.34,0.00),v40,z0,tPen\WObj:=wPaper;
    MoveL Offs(pOrigin,108.05,71.94,0.00),v40,z0,tPen\WObj:=wPaper;
    MoveL Offs(pOrigin,108.26,72.36,0.00),v40,z0,tPen\WObj:=wPaper;
    MoveL Offs(pOrigin,108.05,71.94,0.00),v40,z0,tPen\WObj:=wPaper;
    MoveL Offs(pOrigin,108.37,71.09,0.00),v40,z0,tPen\WObj:=wPaper;
    MoveL Offs(pOrigin,107.02,72.44,0.00),v40,z0,tPen\WObj:=wPaper;
    MoveL Offs(pOrigin,107.77,73.19,0.00),v40,z0,tPen\WObj:=wPaper;
    MoveL Offs(pOrigin,109.12,71.83,0.00),v40,z0,tPen\WObj:=wPaper;
    MoveL Offs(pOrigin,109.71,72.73,0.00),v40,z0,tPen\WObj:=wPaper;
    MoveL Offs(pOrigin,108.36,74.08,0.00),v40,z0,tPen\WObj:=wPaper;
    MoveL Offs(pOrigin,108.96,74.98,0.00),v40,z0,tPen\WObj:=wPaper;
    MoveL Offs(pOrigin,110.46,73.48,0.00),v40,z0,tPen\WObj:=wPaper;
    MoveL Offs(pOrigin,111.06,74.37,0.00),v40,z0,tPen\WObj:=wPaper;
    MoveL Offs(pOrigin,109.56,75.88,0.00),v40,fine,tPen\WObj:=wPaper;
    MoveL Offs(pOrigin,109.56,75.88,6.00),v60,z5,tPen\WObj:=wPaper;
    MoveL Offs(pOrigin,107.75,77.68,6.00),vTravel,z5,tPen\WObj:=wPaper;
    MoveL Offs(pOrigin,107.75,77.68,0.00),v60,z0,tPen\WObj:=wPaper;
    MoveL Offs(pOrigin,106.40,79.03,0.00),v40,z0,tPen\WObj:=wPaper;
    MoveL Offs(pOrigin,106.86,78.78,0.00),v40,z0,tPen\WObj:=wPaper;
    MoveL Offs(pOrigin,114.52,86.44,0.00),v40,z0,tPen\WObj:=wPaper;
    MoveL Offs(pOrigin,113.87,86.50,0.00),v40,z0,tPen\WObj:=wPaper;
    MoveL Offs(pOrigin,115.52,84.85,0.00),v40,z0,tPen\WObj:=wPaper;
    MoveL Offs(pOrigin,114.52,84.94,0.00),v40,z0,tPen\WObj:=wPaper;
    MoveL Offs(pOrigin,118.27,88.70,0.00),v40,z0,tPen\WObj:=wPaper;
    MoveL Offs(pOrigin,118.65,89.18,0.00),v40,z0,tPen\WObj:=wPaper;
    MoveL Offs(pOrigin,120.61,87.23,0.00),v40,z0,tPen\WObj:=wPaper;
    MoveL Offs(pOrigin,120.52,87.96,0.00),v40,z0,tPen\WObj:=wPaper;
    MoveL Offs(pOrigin,122.77,90.21,0.00),v40,z0,tPen\WObj:=wPaper;
    MoveL Offs(pOrigin,121.94,90.37,0.00),v40,z0,tPen\WObj:=wPaper;
    MoveL Offs(pOrigin,124.05,88.27,0.00),v40,z0,tPen\WObj:=wPaper;
    MoveL Offs(pOrigin,124.57,89.02,0.00),v40,z0,tPen\WObj:=wPaper;
    MoveL Offs(pOrigin,128.47,92.92,0.00),v40,z0,tPen\WObj:=wPaper;
    MoveL Offs(pOrigin,129.09,92.09,0.00),v40,z0,tPen\WObj:=wPaper;
    MoveL Offs(pOrigin,124.20,92.09,0.00),v40,z0,tPen\WObj:=wPaper;
    MoveL Offs(pOrigin,124.28,91.71,0.00),v40,z0,tPen\WObj:=wPaper;
    MoveL Offs(pOrigin,126.08,93.52,0.00),v40,z0,tPen\WObj:=wPaper;
    MoveL Offs(pOrigin,125.83,93.95,0.00),v40,z0,tPen\WObj:=wPaper;
    MoveL Offs(pOrigin,131.39,88.39,0.00),v40,z0,tPen\WObj:=wPaper;
    MoveL Offs(pOrigin,132.06,89.04,0.00),v40,z0,tPen\WObj:=wPaper;
    MoveL Offs(pOrigin,133.71,90.69,0.00),v40,z0,tPen\WObj:=wPaper;
    MoveL Offs(pOrigin,134.19,89.98,0.00),v40,z0,tPen\WObj:=wPaper;
    MoveL Offs(pOrigin,129.30,89.98,0.00),v40,z0,tPen\WObj:=wPaper;
    MoveL Offs(pOrigin,129.51,89.48,0.00),v40,z0,tPen\WObj:=wPaper;
    MoveL Offs(pOrigin,131.61,91.59,0.00),v40,z0,tPen\WObj:=wPaper;
    MoveL Offs(pOrigin,131.85,91.03,0.00),v40,z0,tPen\WObj:=wPaper;
    MoveL Offs(pOrigin,127.18,91.03,0.00),v40,z0,tPen\WObj:=wPaper;
    MoveL Offs(pOrigin,127.18,90.00,0.00),v40,z0,tPen\WObj:=wPaper;
    MoveL Offs(pOrigin,128.88,90.07,0.00),v40,z0,tPen\WObj:=wPaper;
    MoveL Offs(pOrigin,133.12,88.87,0.00),v40,z0,tPen\WObj:=wPaper;
    MoveL Offs(pOrigin,133.98,88.30,0.00),v40,z0,tPen\WObj:=wPaper;
    MoveL Offs(pOrigin,134.61,87.31,0.00),v40,z0,tPen\WObj:=wPaper;
    MoveL Offs(pOrigin,136.10,86.88,0.00),v40,z0,tPen\WObj:=wPaper;
    MoveL Offs(pOrigin,139.07,85.32,0.00),v40,z0,tPen\WObj:=wPaper;
    MoveL Offs(pOrigin,139.41,85.11,0.00),v40,z0,tPen\WObj:=wPaper;
    MoveL Offs(pOrigin,139.41,86.39,0.00),v40,z0,tPen\WObj:=wPaper;
    MoveL Offs(pOrigin,139.93,86.81,0.00),v40,z0,tPen\WObj:=wPaper;
  ENDPROC

  PROC DrawPart258()
    MoveL Offs(pOrigin,135.46,86.81,0.00),v40,z0,tPen\WObj:=wPaper;
    MoveL Offs(pOrigin,135.34,86.35,0.00),v40,z0,tPen\WObj:=wPaper;
    MoveL Offs(pOrigin,137.60,88.61,0.00),v40,z0,tPen\WObj:=wPaper;
    MoveL Offs(pOrigin,138.58,88.67,0.00),v40,z0,tPen\WObj:=wPaper;
    MoveL Offs(pOrigin,148.79,78.45,0.00),v40,z0,tPen\WObj:=wPaper;
    MoveL Offs(pOrigin,149.10,79.21,0.00),v40,z0,tPen\WObj:=wPaper;
    MoveL Offs(pOrigin,150.76,80.86,0.00),v40,fine,tPen\WObj:=wPaper;
    MoveL Offs(pOrigin,150.76,80.86,6.00),v60,z5,tPen\WObj:=wPaper;
    MoveL Offs(pOrigin,152.10,80.71,6.00),vTravel,z5,tPen\WObj:=wPaper;
    MoveL Offs(pOrigin,152.10,80.71,0.00),v60,z0,tPen\WObj:=wPaper;
    MoveL Offs(pOrigin,150.15,78.76,0.00),v40,z0,tPen\WObj:=wPaper;
    MoveL Offs(pOrigin,151.20,78.31,0.00),v40,z0,tPen\WObj:=wPaper;
    MoveL Offs(pOrigin,153.15,80.27,0.00),v40,z0,tPen\WObj:=wPaper;
    MoveL Offs(pOrigin,153.28,81.43,0.00),v40,z0,tPen\WObj:=wPaper;
    MoveL Offs(pOrigin,145.17,89.55,0.00),v40,fine,tPen\WObj:=wPaper;
    MoveL Offs(pOrigin,145.17,89.55,6.00),v60,z5,tPen\WObj:=wPaper;
    MoveL Offs(pOrigin,145.99,91.03,6.00),vTravel,z5,tPen\WObj:=wPaper;
    MoveL Offs(pOrigin,145.99,91.03,0.00),v60,z0,tPen\WObj:=wPaper;
    MoveL Offs(pOrigin,146.90,91.93,0.00),v40,z0,tPen\WObj:=wPaper;
    MoveL Offs(pOrigin,146.73,91.49,0.00),v40,z0,tPen\WObj:=wPaper;
    MoveL Offs(pOrigin,146.51,91.70,0.00),v40,z0,tPen\WObj:=wPaper;
    MoveL Offs(pOrigin,146.73,91.28,0.00),v40,z0,tPen\WObj:=wPaper;
    MoveL Offs(pOrigin,147.15,91.28,0.00),v40,z0,tPen\WObj:=wPaper;
    MoveL Offs(pOrigin,147.15,91.28,0.00),v40,z0,tPen\WObj:=wPaper;
    MoveL Offs(pOrigin,148.21,91.06,0.00),v40,z0,tPen\WObj:=wPaper;
    MoveL Offs(pOrigin,148.43,90.43,0.00),v40,z0,tPen\WObj:=wPaper;
    MoveL Offs(pOrigin,148.43,90.43,0.00),v40,z0,tPen\WObj:=wPaper;
    MoveL Offs(pOrigin,149.20,90.14,0.00),v40,z0,tPen\WObj:=wPaper;
    MoveL Offs(pOrigin,149.27,89.43,0.00),v40,z0,tPen\WObj:=wPaper;
    MoveL Offs(pOrigin,148.43,89.57,0.00),v40,z0,tPen\WObj:=wPaper;
    MoveL Offs(pOrigin,148.21,90.21,0.00),v40,z0,tPen\WObj:=wPaper;
    MoveL Offs(pOrigin,148.21,90.21,0.00),v40,z0,tPen\WObj:=wPaper;
    MoveL Offs(pOrigin,147.57,90.21,0.00),v40,z0,tPen\WObj:=wPaper;
    MoveL Offs(pOrigin,147.15,90.64,0.00),v40,z0,tPen\WObj:=wPaper;
    MoveL Offs(pOrigin,147.15,91.28,0.00),v40,z0,tPen\WObj:=wPaper;
    MoveL Offs(pOrigin,147.79,91.34,0.00),v40,z0,tPen\WObj:=wPaper;
    MoveL Offs(pOrigin,146.89,90.43,0.00),v40,z0,tPen\WObj:=wPaper;
    MoveL Offs(pOrigin,147.79,89.84,0.00),v40,z0,tPen\WObj:=wPaper;
    MoveL Offs(pOrigin,148.69,90.74,0.00),v40,z0,tPen\WObj:=wPaper;
    MoveL Offs(pOrigin,149.59,90.14,0.00),v40,z0,tPen\WObj:=wPaper;
    MoveL Offs(pOrigin,148.53,89.09,0.00),v40,z0,tPen\WObj:=wPaper;
    MoveL Offs(pOrigin,149.49,89.36,0.00),v40,z0,tPen\WObj:=wPaper;
    MoveL Offs(pOrigin,153.52,85.32,0.00),v40,z0,tPen\WObj:=wPaper;
    MoveL Offs(pOrigin,156.36,81.50,0.00),v40,z0,tPen\WObj:=wPaper;
    MoveL Offs(pOrigin,157.14,79.80,0.00),v40,fine,tPen\WObj:=wPaper;
    MoveL Offs(pOrigin,157.14,79.80,6.00),v60,z5,tPen\WObj:=wPaper;
    MoveL Offs(pOrigin,155.10,79.22,6.00),vTravel,z5,tPen\WObj:=wPaper;
    MoveL Offs(pOrigin,155.10,79.22,0.00),v60,z0,tPen\WObj:=wPaper;
    MoveL Offs(pOrigin,153.44,77.57,0.00),v40,fine,tPen\WObj:=wPaper;
    MoveL Offs(pOrigin,153.44,77.57,6.00),v60,z5,tPen\WObj:=wPaper;
    MoveL Offs(pOrigin,154.03,82.18,6.00),vTravel,z5,tPen\WObj:=wPaper;
    MoveL Offs(pOrigin,154.03,82.18,0.00),v60,z0,tPen\WObj:=wPaper;
    MoveL Offs(pOrigin,168.60,67.61,0.00),v40,z0,tPen\WObj:=wPaper;
    MoveL Offs(pOrigin,169.50,68.20,0.00),v40,z0,tPen\WObj:=wPaper;
    MoveL Offs(pOrigin,143.05,94.65,0.00),v40,fine,tPen\WObj:=wPaper;
    MoveL Offs(pOrigin,143.05,94.65,6.00),v60,z5,tPen\WObj:=wPaper;
    MoveL Offs(pOrigin,144.05,93.57,6.00),vTravel,z5,tPen\WObj:=wPaper;
    MoveL Offs(pOrigin,144.05,93.57,0.00),v60,z0,tPen\WObj:=wPaper;
    MoveL Offs(pOrigin,143.30,92.82,0.00),v40,z0,tPen\WObj:=wPaper;
    MoveL Offs(pOrigin,142.76,91.95,0.00),v40,z0,tPen\WObj:=wPaper;
    MoveL Offs(pOrigin,138.55,96.16,0.00),v40,fine,tPen\WObj:=wPaper;
    MoveL Offs(pOrigin,138.55,96.16,6.00),v60,z5,tPen\WObj:=wPaper;
    MoveL Offs(pOrigin,136.91,96.32,6.00),vTravel,z5,tPen\WObj:=wPaper;
    MoveL Offs(pOrigin,136.91,96.32,0.00),v60,z0,tPen\WObj:=wPaper;
    MoveL Offs(pOrigin,139.76,93.46,0.00),v40,fine,tPen\WObj:=wPaper;
    MoveL Offs(pOrigin,139.76,93.46,6.00),v60,z5,tPen\WObj:=wPaper;
    MoveL Offs(pOrigin,140.80,95.40,6.00),vTravel,z5,tPen\WObj:=wPaper;
    MoveL Offs(pOrigin,140.80,95.40,0.00),v60,z0,tPen\WObj:=wPaper;
    MoveL Offs(pOrigin,147.41,88.79,0.00),v40,fine,tPen\WObj:=wPaper;
    MoveL Offs(pOrigin,147.41,88.79,6.00),v60,z5,tPen\WObj:=wPaper;
    MoveL Offs(pOrigin,149.43,88.49,6.00),vTravel,z5,tPen\WObj:=wPaper;
    MoveL Offs(pOrigin,149.43,88.49,0.00),v60,z0,tPen\WObj:=wPaper;
    MoveL Offs(pOrigin,150.33,89.40,0.00),v40,z0,tPen\WObj:=wPaper;
    MoveL Offs(pOrigin,151.23,88.80,0.00),v40,z0,tPen\WObj:=wPaper;
    MoveL Offs(pOrigin,150.33,87.90,0.00),v40,z0,tPen\WObj:=wPaper;
    MoveL Offs(pOrigin,150.92,87.00,0.00),v40,z0,tPen\WObj:=wPaper;
    MoveL Offs(pOrigin,151.83,87.90,0.00),v40,z0,tPen\WObj:=wPaper;
    MoveL Offs(pOrigin,152.57,87.16,0.00),v40,z0,tPen\WObj:=wPaper;
    MoveL Offs(pOrigin,151.67,86.25,0.00),v40,z0,tPen\WObj:=wPaper;
    MoveL Offs(pOrigin,152.04,86.81,0.00),v40,z0,tPen\WObj:=wPaper;
    MoveL Offs(pOrigin,150.55,88.30,0.00),v40,z0,tPen\WObj:=wPaper;
    MoveL Offs(pOrigin,152.04,86.81,0.00),v40,fine,tPen\WObj:=wPaper;
    MoveL Offs(pOrigin,152.04,86.81,6.00),v60,z5,tPen\WObj:=wPaper;
    MoveL Offs(pOrigin,153.32,86.41,6.00),vTravel,z5,tPen\WObj:=wPaper;
    MoveL Offs(pOrigin,153.32,86.41,0.00),v60,z0,tPen\WObj:=wPaper;
    MoveL Offs(pOrigin,152.42,85.51,0.00),v40,z0,tPen\WObj:=wPaper;
    MoveL Offs(pOrigin,153.16,84.76,0.00),v40,z0,tPen\WObj:=wPaper;
    MoveL Offs(pOrigin,153.92,85.51,0.00),v40,z0,tPen\WObj:=wPaper;
    MoveL Offs(pOrigin,153.52,85.11,0.00),v40,z0,tPen\WObj:=wPaper;
    MoveL Offs(pOrigin,152.46,86.18,0.00),v40,z0,tPen\WObj:=wPaper;
    MoveL Offs(pOrigin,153.52,85.11,0.00),v40,fine,tPen\WObj:=wPaper;
    MoveL Offs(pOrigin,153.52,85.11,6.00),v60,z5,tPen\WObj:=wPaper;
    MoveL Offs(pOrigin,151.61,81.93,6.00),vTravel,z5,tPen\WObj:=wPaper;
    MoveL Offs(pOrigin,151.61,81.93,0.00),v60,z0,tPen\WObj:=wPaper;
    MoveL Offs(pOrigin,150.98,82.56,0.00),v40,z0,tPen\WObj:=wPaper;
    MoveL Offs(pOrigin,151.61,81.93,0.00),v40,fine,tPen\WObj:=wPaper;
    MoveL Offs(pOrigin,151.61,81.93,6.00),v60,z5,tPen\WObj:=wPaper;
    MoveL Offs(pOrigin,150.05,83.77,6.00),vTravel,z5,tPen\WObj:=wPaper;
    MoveL Offs(pOrigin,150.05,83.77,0.00),v60,z0,tPen\WObj:=wPaper;
    MoveL Offs(pOrigin,146.09,87.66,0.00),v40,z0,tPen\WObj:=wPaper;
    MoveL Offs(pOrigin,150.05,83.77,0.00),v40,fine,tPen\WObj:=wPaper;
    MoveL Offs(pOrigin,150.05,83.77,6.00),v60,z5,tPen\WObj:=wPaper;
    MoveL Offs(pOrigin,148.43,81.50,6.00),vTravel,z5,tPen\WObj:=wPaper;
    MoveL Offs(pOrigin,148.43,81.50,0.00),v60,z0,tPen\WObj:=wPaper;
    MoveL Offs(pOrigin,148.85,81.29,0.00),v40,z0,tPen\WObj:=wPaper;
    MoveL Offs(pOrigin,148.43,81.50,0.00),v40,z0,tPen\WObj:=wPaper;
    MoveL Offs(pOrigin,148.00,81.71,0.00),v40,z0,tPen\WObj:=wPaper;
    MoveL Offs(pOrigin,150.55,80.37,0.00),v40,z0,tPen\WObj:=wPaper;
    MoveL Offs(pOrigin,152.25,79.80,0.00),v40,z0,tPen\WObj:=wPaper;
    MoveL Offs(pOrigin,153.52,79.80,0.00),v40,z0,tPen\WObj:=wPaper;
    MoveL Offs(pOrigin,154.02,79.23,0.00),v40,z0,tPen\WObj:=wPaper;
    MoveL Offs(pOrigin,157.77,78.10,0.00),v40,z0,tPen\WObj:=wPaper;
    MoveL Offs(pOrigin,158.27,78.31,0.00),v40,z0,tPen\WObj:=wPaper;
    MoveL Offs(pOrigin,159.90,83.62,0.00),v40,z0,tPen\WObj:=wPaper;
    MoveL Offs(pOrigin,160.32,86.81,0.00),v40,z0,tPen\WObj:=wPaper;
    MoveL Offs(pOrigin,160.32,91.06,0.00),v40,z0,tPen\WObj:=wPaper;
    MoveL Offs(pOrigin,157.99,90.64,0.00),v40,z0,tPen\WObj:=wPaper;
    MoveL Offs(pOrigin,155.23,91.84,0.00),v40,z0,tPen\WObj:=wPaper;
    MoveL Offs(pOrigin,154.52,92.76,0.00),v40,z0,tPen\WObj:=wPaper;
    MoveL Offs(pOrigin,154.80,92.97,0.00),v40,z0,tPen\WObj:=wPaper;
  ENDPROC

  PROC DrawPart259()
    MoveL Offs(pOrigin,157.35,91.91,0.00),v40,z0,tPen\WObj:=wPaper;
    MoveL Offs(pOrigin,159.05,92.20,0.00),v40,z0,tPen\WObj:=wPaper;
    MoveL Offs(pOrigin,160.54,93.40,0.00),v40,z0,tPen\WObj:=wPaper;
    MoveL Offs(pOrigin,161.95,95.53,0.00),v40,z0,tPen\WObj:=wPaper;
    MoveL Offs(pOrigin,162.45,97.01,0.00),v40,z0,tPen\WObj:=wPaper;
    MoveL Offs(pOrigin,162.66,99.35,0.00),v40,z0,tPen\WObj:=wPaper;
    MoveL Offs(pOrigin,162.02,100.41,0.00),v40,z0,tPen\WObj:=wPaper;
    MoveL Offs(pOrigin,162.02,100.41,0.00),v40,z0,tPen\WObj:=wPaper;
    MoveL Offs(pOrigin,161.18,99.99,0.00),v40,fine,tPen\WObj:=wPaper;
    MoveL Offs(pOrigin,161.18,99.99,6.00),v60,z5,tPen\WObj:=wPaper;
    MoveL Offs(pOrigin,162.64,100.62,6.00),vTravel,z5,tPen\WObj:=wPaper;
    MoveL Offs(pOrigin,162.64,100.62,0.00),v60,z0,tPen\WObj:=wPaper;
    MoveL Offs(pOrigin,162.64,110.19,0.00),v40,z0,tPen\WObj:=wPaper;
    MoveL Offs(pOrigin,162.88,111.10,0.00),v40,z0,tPen\WObj:=wPaper;
    MoveL Offs(pOrigin,160.75,111.10,0.00),v40,z0,tPen\WObj:=wPaper;
    MoveL Offs(pOrigin,160.75,112.15,0.00),v40,z0,tPen\WObj:=wPaper;
    MoveL Offs(pOrigin,162.66,112.15,0.00),v40,fine,tPen\WObj:=wPaper;
    MoveL Offs(pOrigin,162.66,112.15,6.00),v60,z5,tPen\WObj:=wPaper;
    MoveL Offs(pOrigin,160.14,112.65,6.00),vTravel,z5,tPen\WObj:=wPaper;
    MoveL Offs(pOrigin,160.14,112.65,0.00),v60,z0,tPen\WObj:=wPaper;
    MoveL Offs(pOrigin,162.55,115.05,0.00),v40,z0,tPen\WObj:=wPaper;
    MoveL Offs(pOrigin,163.06,114.96,0.00),v40,z0,tPen\WObj:=wPaper;
    MoveL Offs(pOrigin,158.10,119.92,0.00),v40,z0,tPen\WObj:=wPaper;
    MoveL Offs(pOrigin,158.20,119.54,0.00),v40,z0,tPen\WObj:=wPaper;
    MoveL Offs(pOrigin,155.44,119.96,0.00),v40,z0,tPen\WObj:=wPaper;
    MoveL Offs(pOrigin,152.25,119.96,0.00),v40,z0,tPen\WObj:=wPaper;
    MoveL Offs(pOrigin,152.25,119.96,0.00),v40,z0,tPen\WObj:=wPaper;
    MoveL Offs(pOrigin,151.82,119.32,0.00),v40,z0,tPen\WObj:=wPaper;
    MoveL Offs(pOrigin,150.34,119.32,0.00),v40,z0,tPen\WObj:=wPaper;
    MoveL Offs(pOrigin,150.34,119.32,0.00),v40,z0,tPen\WObj:=wPaper;
    MoveL Offs(pOrigin,149.27,119.11,0.00),v40,z0,tPen\WObj:=wPaper;
    MoveL Offs(pOrigin,149.06,119.75,0.00),v40,z0,tPen\WObj:=wPaper;
    MoveL Offs(pOrigin,149.06,119.75,0.00),v40,z0,tPen\WObj:=wPaper;
    MoveL Offs(pOrigin,147.79,119.54,0.00),v40,z0,tPen\WObj:=wPaper;
    MoveL Offs(pOrigin,147.79,119.54,0.00),v40,z0,tPen\WObj:=wPaper;
    MoveL Offs(pOrigin,148.00,118.90,0.00),v40,z0,tPen\WObj:=wPaper;
    MoveL Offs(pOrigin,149.06,119.11,0.00),v40,z0,tPen\WObj:=wPaper;
    MoveL Offs(pOrigin,149.06,119.75,0.00),v40,z0,tPen\WObj:=wPaper;
    MoveL Offs(pOrigin,150.34,119.96,0.00),v40,z0,tPen\WObj:=wPaper;
    MoveL Offs(pOrigin,149.83,120.25,0.00),v40,z0,tPen\WObj:=wPaper;
    MoveL Offs(pOrigin,148.18,118.60,0.00),v40,z0,tPen\WObj:=wPaper;
    MoveL Offs(pOrigin,147.79,118.90,0.00),v40,z0,tPen\WObj:=wPaper;
    MoveL Offs(pOrigin,147.57,118.69,0.00),v40,z0,tPen\WObj:=wPaper;
    MoveL Offs(pOrigin,146.73,118.90,0.00),v40,z0,tPen\WObj:=wPaper;
    MoveL Offs(pOrigin,146.73,118.90,0.00),v40,z0,tPen\WObj:=wPaper;
    MoveL Offs(pOrigin,147.15,119.54,0.00),v40,z0,tPen\WObj:=wPaper;
    MoveL Offs(pOrigin,147.79,119.54,0.00),v40,z0,tPen\WObj:=wPaper;
    MoveL Offs(pOrigin,148.18,120.10,0.00),v40,z0,tPen\WObj:=wPaper;
    MoveL Offs(pOrigin,146.38,118.30,0.00),v40,z0,tPen\WObj:=wPaper;
    MoveL Offs(pOrigin,146.73,118.90,0.00),v40,z0,tPen\WObj:=wPaper;
    MoveL Offs(pOrigin,144.39,118.47,0.00),v40,z0,tPen\WObj:=wPaper;
    MoveL Offs(pOrigin,137.38,116.14,0.00),v40,fine,tPen\WObj:=wPaper;
    MoveL Offs(pOrigin,137.38,116.14,6.00),v60,z5,tPen\WObj:=wPaper;
    MoveL Offs(pOrigin,138.64,116.98,6.00),vTravel,z5,tPen\WObj:=wPaper;
    MoveL Offs(pOrigin,138.64,116.98,0.00),v60,z0,tPen\WObj:=wPaper;
    MoveL Offs(pOrigin,139.54,116.08,0.00),v40,fine,tPen\WObj:=wPaper;
    MoveL Offs(pOrigin,139.54,116.08,6.00),v60,z5,tPen\WObj:=wPaper;
    MoveL Offs(pOrigin,140.74,116.38,6.00),vTravel,z5,tPen\WObj:=wPaper;
    MoveL Offs(pOrigin,140.74,116.38,0.00),v60,z0,tPen\WObj:=wPaper;
    MoveL Offs(pOrigin,139.54,117.58,0.00),v40,z0,tPen\WObj:=wPaper;
    MoveL Offs(pOrigin,140.58,118.02,0.00),v40,z0,tPen\WObj:=wPaper;
    MoveL Offs(pOrigin,141.94,116.67,0.00),v40,fine,tPen\WObj:=wPaper;
    MoveL Offs(pOrigin,141.94,116.67,6.00),v60,z5,tPen\WObj:=wPaper;
    MoveL Offs(pOrigin,143.13,116.97,6.00),vTravel,z5,tPen\WObj:=wPaper;
    MoveL Offs(pOrigin,143.13,116.97,0.00),v60,z0,tPen\WObj:=wPaper;
    MoveL Offs(pOrigin,141.63,118.47,0.00),v40,z0,tPen\WObj:=wPaper;
    MoveL Offs(pOrigin,142.68,118.92,0.00),v40,z0,tPen\WObj:=wPaper;
    MoveL Offs(pOrigin,144.48,117.11,0.00),v40,z0,tPen\WObj:=wPaper;
    MoveL Offs(pOrigin,144.73,118.14,0.00),v40,z0,tPen\WObj:=wPaper;
    MoveL Offs(pOrigin,146.23,119.64,0.00),v40,z0,tPen\WObj:=wPaper;
    MoveL Offs(pOrigin,146.12,119.96,0.00),v40,z0,tPen\WObj:=wPaper;
    MoveL Offs(pOrigin,150.93,115.15,0.00),v40,z0,tPen\WObj:=wPaper;
    MoveL Offs(pOrigin,151.31,115.76,0.00),v40,z0,tPen\WObj:=wPaper;
    MoveL Offs(pOrigin,153.27,117.72,0.00),v40,fine,tPen\WObj:=wPaper;
    MoveL Offs(pOrigin,153.27,117.72,6.00),v60,z5,tPen\WObj:=wPaper;
    MoveL Offs(pOrigin,154.76,117.72,6.00),vTravel,z5,tPen\WObj:=wPaper;
    MoveL Offs(pOrigin,154.76,117.72,0.00),v60,z0,tPen\WObj:=wPaper;
    MoveL Offs(pOrigin,152.81,115.77,0.00),v40,z0,tPen\WObj:=wPaper;
    MoveL Offs(pOrigin,152.43,115.14,0.00),v40,z0,tPen\WObj:=wPaper;
    MoveL Offs(pOrigin,147.32,120.25,0.00),v40,fine,tPen\WObj:=wPaper;
    MoveL Offs(pOrigin,147.32,120.25,6.00),v60,z5,tPen\WObj:=wPaper;
    MoveL Offs(pOrigin,148.52,120.55,6.00),vTravel,z5,tPen\WObj:=wPaper;
    MoveL Offs(pOrigin,148.52,120.55,0.00),v60,z0,tPen\WObj:=wPaper;
    MoveL Offs(pOrigin,153.93,115.14,0.00),v40,z0,tPen\WObj:=wPaper;
    MoveL Offs(pOrigin,154.31,115.77,0.00),v40,z0,tPen\WObj:=wPaper;
    MoveL Offs(pOrigin,156.11,117.58,0.00),v40,z0,tPen\WObj:=wPaper;
    MoveL Offs(pOrigin,156.46,118.58,0.00),v40,z0,tPen\WObj:=wPaper;
    MoveL Offs(pOrigin,154.06,120.98,0.00),v40,z0,tPen\WObj:=wPaper;
    MoveL Offs(pOrigin,154.62,120.57,0.00),v40,z0,tPen\WObj:=wPaper;
    MoveL Offs(pOrigin,153.42,119.37,0.00),v40,fine,tPen\WObj:=wPaper;
    MoveL Offs(pOrigin,153.42,119.37,6.00),v60,z5,tPen\WObj:=wPaper;
    MoveL Offs(pOrigin,153.12,120.56,6.00),vTravel,z5,tPen\WObj:=wPaper;
    MoveL Offs(pOrigin,153.12,120.56,0.00),v60,z0,tPen\WObj:=wPaper;
    MoveL Offs(pOrigin,151.77,119.21,0.00),v40,z0,tPen\WObj:=wPaper;
    MoveL Offs(pOrigin,152.25,119.96,0.00),v40,z0,tPen\WObj:=wPaper;
    MoveL Offs(pOrigin,150.76,120.18,0.00),v40,z0,tPen\WObj:=wPaper;
    MoveL Offs(pOrigin,150.34,119.32,0.00),v40,z0,tPen\WObj:=wPaper;
    MoveL Offs(pOrigin,149.97,118.91,0.00),v40,z0,tPen\WObj:=wPaper;
    MoveL Offs(pOrigin,151.63,120.56,0.00),v40,z0,tPen\WObj:=wPaper;
    MoveL Offs(pOrigin,151.21,120.84,0.00),v40,z0,tPen\WObj:=wPaper;
    MoveL Offs(pOrigin,165.94,106.11,0.00),v40,z0,tPen\WObj:=wPaper;
    MoveL Offs(pOrigin,165.34,105.22,0.00),v40,z0,tPen\WObj:=wPaper;
    MoveL Offs(pOrigin,158.73,111.83,0.00),v40,z0,tPen\WObj:=wPaper;
    MoveL Offs(pOrigin,158.79,111.29,0.00),v40,z0,tPen\WObj:=wPaper;
    MoveL Offs(pOrigin,157.44,109.94,0.00),v40,z0,tPen\WObj:=wPaper;
    MoveL Offs(pOrigin,158.14,109.43,0.00),v40,z0,tPen\WObj:=wPaper;
    MoveL Offs(pOrigin,155.43,112.14,0.00),v40,z0,tPen\WObj:=wPaper;
    MoveL Offs(pOrigin,154.90,111.88,0.00),v40,z0,tPen\WObj:=wPaper;
    MoveL Offs(pOrigin,153.24,110.23,0.00),v40,z0,tPen\WObj:=wPaper;
    MoveL Offs(pOrigin,153.34,109.75,0.00),v40,z0,tPen\WObj:=wPaper;
    MoveL Offs(pOrigin,150.34,112.75,0.00),v40,z0,tPen\WObj:=wPaper;
    MoveL Offs(pOrigin,150.85,112.32,0.00),v40,z0,tPen\WObj:=wPaper;
    MoveL Offs(pOrigin,149.50,110.96,0.00),v40,z0,tPen\WObj:=wPaper;
    MoveL Offs(pOrigin,150.05,110.06,0.00),v40,z0,tPen\WObj:=wPaper;
    MoveL Offs(pOrigin,146.89,113.21,0.00),v40,z0,tPen\WObj:=wPaper;
    MoveL Offs(pOrigin,146.66,112.60,0.00),v40,z0,tPen\WObj:=wPaper;
    MoveL Offs(pOrigin,145.16,111.10,0.00),v40,z0,tPen\WObj:=wPaper;
    MoveL Offs(pOrigin,145.10,110.52,0.00),v40,z0,tPen\WObj:=wPaper;
    MoveL Offs(pOrigin,142.25,113.38,0.00),v40,z0,tPen\WObj:=wPaper;
    MoveL Offs(pOrigin,142.47,112.89,0.00),v40,z0,tPen\WObj:=wPaper;
  ENDPROC

  PROC DrawPart260()
    MoveL Offs(pOrigin,141.11,111.54,0.00),v40,z0,tPen\WObj:=wPaper;
    MoveL Offs(pOrigin,141.80,110.83,0.00),v40,z0,tPen\WObj:=wPaper;
    MoveL Offs(pOrigin,139.25,113.39,0.00),v40,z0,tPen\WObj:=wPaper;
    MoveL Offs(pOrigin,139.62,113.03,0.00),v40,z0,tPen\WObj:=wPaper;
    MoveL Offs(pOrigin,138.27,111.68,0.00),v40,z0,tPen\WObj:=wPaper;
    MoveL Offs(pOrigin,138.81,110.84,0.00),v40,z0,tPen\WObj:=wPaper;
    MoveL Offs(pOrigin,136.40,113.24,0.00),v40,z0,tPen\WObj:=wPaper;
    MoveL Offs(pOrigin,136.47,112.87,0.00),v40,z0,tPen\WObj:=wPaper;
    MoveL Offs(pOrigin,135.27,111.67,0.00),v40,z0,tPen\WObj:=wPaper;
    MoveL Offs(pOrigin,135.81,110.85,0.00),v40,z0,tPen\WObj:=wPaper;
    MoveL Offs(pOrigin,133.56,113.10,0.00),v40,fine,tPen\WObj:=wPaper;
    MoveL Offs(pOrigin,133.56,113.10,6.00),v60,z5,tPen\WObj:=wPaper;
    MoveL Offs(pOrigin,132.36,112.81,6.00),vTravel,z5,tPen\WObj:=wPaper;
    MoveL Offs(pOrigin,132.36,112.81,0.00),v60,z0,tPen\WObj:=wPaper;
    MoveL Offs(pOrigin,134.01,111.15,0.00),v40,z0,tPen\WObj:=wPaper;
    MoveL Offs(pOrigin,134.07,111.97,0.00),v40,z0,tPen\WObj:=wPaper;
    MoveL Offs(pOrigin,134.98,112.87,0.00),v40,z0,tPen\WObj:=wPaper;
    MoveL Offs(pOrigin,134.91,113.25,0.00),v40,z0,tPen\WObj:=wPaper;
    MoveL Offs(pOrigin,137.31,110.84,0.00),v40,z0,tPen\WObj:=wPaper;
    MoveL Offs(pOrigin,136.77,111.67,0.00),v40,z0,tPen\WObj:=wPaper;
    MoveL Offs(pOrigin,138.12,113.03,0.00),v40,z0,tPen\WObj:=wPaper;
    MoveL Offs(pOrigin,137.75,113.39,0.00),v40,z0,tPen\WObj:=wPaper;
    MoveL Offs(pOrigin,140.16,110.99,0.00),v40,z0,tPen\WObj:=wPaper;
    MoveL Offs(pOrigin,139.62,111.53,0.00),v40,z0,tPen\WObj:=wPaper;
    MoveL Offs(pOrigin,140.97,112.89,0.00),v40,z0,tPen\WObj:=wPaper;
    MoveL Offs(pOrigin,140.75,113.38,0.00),v40,z0,tPen\WObj:=wPaper;
    MoveL Offs(pOrigin,143.60,110.53,0.00),v40,z0,tPen\WObj:=wPaper;
    MoveL Offs(pOrigin,143.96,111.40,0.00),v40,z0,tPen\WObj:=wPaper;
    MoveL Offs(pOrigin,145.46,112.90,0.00),v40,z0,tPen\WObj:=wPaper;
    MoveL Offs(pOrigin,145.24,113.37,0.00),v40,z0,tPen\WObj:=wPaper;
    MoveL Offs(pOrigin,148.25,110.36,0.00),v40,z0,tPen\WObj:=wPaper;
    MoveL Offs(pOrigin,148.00,110.96,0.00),v40,z0,tPen\WObj:=wPaper;
    MoveL Offs(pOrigin,149.50,112.46,0.00),v40,z0,tPen\WObj:=wPaper;
    MoveL Offs(pOrigin,148.69,112.91,0.00),v40,z0,tPen\WObj:=wPaper;
    MoveL Offs(pOrigin,151.84,109.75,0.00),v40,z0,tPen\WObj:=wPaper;
    MoveL Offs(pOrigin,152.05,110.52,0.00),v40,z0,tPen\WObj:=wPaper;
    MoveL Offs(pOrigin,153.55,112.03,0.00),v40,z0,tPen\WObj:=wPaper;
    MoveL Offs(pOrigin,153.78,112.29,0.00),v40,z0,tPen\WObj:=wPaper;
    MoveL Offs(pOrigin,156.64,109.44,0.00),v40,z0,tPen\WObj:=wPaper;
    MoveL Offs(pOrigin,156.09,110.09,0.00),v40,z0,tPen\WObj:=wPaper;
    MoveL Offs(pOrigin,157.59,111.59,0.00),v40,z0,tPen\WObj:=wPaper;
    MoveL Offs(pOrigin,156.93,112.13,0.00),v40,z0,tPen\WObj:=wPaper;
    MoveL Offs(pOrigin,159.63,109.43,0.00),v40,z0,tPen\WObj:=wPaper;
    MoveL Offs(pOrigin,160.39,108.68,0.00),v40,z0,tPen\WObj:=wPaper;
    MoveL Offs(pOrigin,165.19,103.87,0.00),v40,fine,tPen\WObj:=wPaper;
    MoveL Offs(pOrigin,165.19,103.87,6.00),v60,z5,tPen\WObj:=wPaper;
    MoveL Offs(pOrigin,164.36,104.76,6.00),vTravel,z5,tPen\WObj:=wPaper;
    MoveL Offs(pOrigin,164.36,104.76,0.00),v60,z0,tPen\WObj:=wPaper;
    MoveL Offs(pOrigin,158.20,104.76,0.00),v40,z0,tPen\WObj:=wPaper;
    MoveL Offs(pOrigin,157.87,104.40,0.00),v40,z0,tPen\WObj:=wPaper;
    MoveL Offs(pOrigin,159.52,106.05,0.00),v40,fine,tPen\WObj:=wPaper;
    MoveL Offs(pOrigin,159.52,106.05,6.00),v60,z5,tPen\WObj:=wPaper;
    MoveL Offs(pOrigin,158.32,106.35,6.00),vTravel,z5,tPen\WObj:=wPaper;
    MoveL Offs(pOrigin,158.32,106.35,0.00),v60,z0,tPen\WObj:=wPaper;
    MoveL Offs(pOrigin,156.82,104.85,0.00),v40,z0,tPen\WObj:=wPaper;
    MoveL Offs(pOrigin,156.50,105.82,0.00),v40,z0,tPen\WObj:=wPaper;
    MoveL Offs(pOrigin,158.20,105.82,0.00),v40,fine,tPen\WObj:=wPaper;
    MoveL Offs(pOrigin,158.20,105.82,6.00),v60,z5,tPen\WObj:=wPaper;
    MoveL Offs(pOrigin,157.28,106.79,6.00),vTravel,z5,tPen\WObj:=wPaper;
    MoveL Offs(pOrigin,157.28,106.79,0.00),v60,z0,tPen\WObj:=wPaper;
    MoveL Offs(pOrigin,155.92,105.44,0.00),v40,z0,tPen\WObj:=wPaper;
    MoveL Offs(pOrigin,155.03,106.04,0.00),v40,z0,tPen\WObj:=wPaper;
    MoveL Offs(pOrigin,156.08,107.09,0.00),v40,fine,tPen\WObj:=wPaper;
    MoveL Offs(pOrigin,156.08,107.09,6.00),v60,z5,tPen\WObj:=wPaper;
    MoveL Offs(pOrigin,154.88,107.39,6.00),vTravel,z5,tPen\WObj:=wPaper;
    MoveL Offs(pOrigin,154.88,107.39,0.00),v60,z0,tPen\WObj:=wPaper;
    MoveL Offs(pOrigin,153.98,106.48,0.00),v40,z0,tPen\WObj:=wPaper;
    MoveL Offs(pOrigin,154.16,107.21,0.00),v40,z0,tPen\WObj:=wPaper;
    MoveL Offs(pOrigin,149.49,108.06,0.00),v40,z0,tPen\WObj:=wPaper;
    MoveL Offs(pOrigin,150.35,108.26,0.00),v40,z0,tPen\WObj:=wPaper;
    MoveL Offs(pOrigin,152.30,106.30,0.00),v40,z0,tPen\WObj:=wPaper;
    MoveL Offs(pOrigin,152.93,106.93,0.00),v40,z0,tPen\WObj:=wPaper;
    MoveL Offs(pOrigin,153.83,107.83,0.00),v40,z0,tPen\WObj:=wPaper;
    MoveL Offs(pOrigin,153.05,108.55,0.00),v40,z0,tPen\WObj:=wPaper;
    MoveL Offs(pOrigin,157.85,103.74,0.00),v40,fine,tPen\WObj:=wPaper;
    MoveL Offs(pOrigin,157.85,103.74,6.00),v60,z5,tPen\WObj:=wPaper;
    MoveL Offs(pOrigin,157.39,107.19,6.00),vTravel,z5,tPen\WObj:=wPaper;
    MoveL Offs(pOrigin,157.39,107.19,0.00),v60,z0,tPen\WObj:=wPaper;
    MoveL Offs(pOrigin,165.21,99.37,0.00),v40,fine,tPen\WObj:=wPaper;
    MoveL Offs(pOrigin,165.21,99.37,6.00),v60,z5,tPen\WObj:=wPaper;
    MoveL Offs(pOrigin,163.69,99.99,6.00),vTravel,z5,tPen\WObj:=wPaper;
    MoveL Offs(pOrigin,163.69,99.99,0.00),v60,z0,tPen\WObj:=wPaper;
    MoveL Offs(pOrigin,163.69,95.74,0.00),v40,z0,tPen\WObj:=wPaper;
    MoveL Offs(pOrigin,164.75,95.74,0.00),v40,z0,tPen\WObj:=wPaper;
    MoveL Offs(pOrigin,164.75,96.80,0.00),v40,z0,tPen\WObj:=wPaper;
    MoveL Offs(pOrigin,165.00,97.37,0.00),v40,z0,tPen\WObj:=wPaper;
    MoveL Offs(pOrigin,162.66,97.37,0.00),v40,fine,tPen\WObj:=wPaper;
    MoveL Offs(pOrigin,162.66,97.37,6.00),v60,z5,tPen\WObj:=wPaper;
    MoveL Offs(pOrigin,161.17,95.94,6.00),vTravel,z5,tPen\WObj:=wPaper;
    MoveL Offs(pOrigin,161.17,95.94,0.00),v60,z0,tPen\WObj:=wPaper;
    MoveL Offs(pOrigin,174.25,82.87,0.00),v40,fine,tPen\WObj:=wPaper;
    MoveL Offs(pOrigin,174.25,82.87,6.00),v60,z5,tPen\WObj:=wPaper;
    MoveL Offs(pOrigin,178.39,80.47,6.00),vTravel,z5,tPen\WObj:=wPaper;
    MoveL Offs(pOrigin,178.39,80.47,0.00),v60,z0,tPen\WObj:=wPaper;
    MoveL Offs(pOrigin,180.51,80.47,0.00),v40,z0,tPen\WObj:=wPaper;
    MoveL Offs(pOrigin,181.15,80.65,0.00),v40,z0,tPen\WObj:=wPaper;
    MoveL Offs(pOrigin,181.36,80.01,0.00),v40,z0,tPen\WObj:=wPaper;
    MoveL Offs(pOrigin,183.27,78.45,0.00),v40,z0,tPen\WObj:=wPaper;
    MoveL Offs(pOrigin,184.55,77.89,0.00),v40,z0,tPen\WObj:=wPaper;
    MoveL Offs(pOrigin,185.61,78.31,0.00),v40,fine,tPen\WObj:=wPaper;
    MoveL Offs(pOrigin,185.61,78.31,6.00),v60,z5,tPen\WObj:=wPaper;
    MoveL Offs(pOrigin,185.21,79.47,6.00),vTravel,z5,tPen\WObj:=wPaper;
    MoveL Offs(pOrigin,185.21,79.47,0.00),v60,z0,tPen\WObj:=wPaper;
    MoveL Offs(pOrigin,182.35,76.61,0.00),v40,z0,tPen\WObj:=wPaper;
    MoveL Offs(pOrigin,181.65,77.46,0.00),v40,z0,tPen\WObj:=wPaper;
    MoveL Offs(pOrigin,181.65,78.95,0.00),v40,z0,tPen\WObj:=wPaper;
    MoveL Offs(pOrigin,181.79,79.42,0.00),v40,z0,tPen\WObj:=wPaper;
    MoveL Offs(pOrigin,179.45,79.42,0.00),v40,z0,tPen\WObj:=wPaper;
    MoveL Offs(pOrigin,179.66,79.16,0.00),v40,z0,tPen\WObj:=wPaper;
    MoveL Offs(pOrigin,179.45,79.59,0.00),v40,z0,tPen\WObj:=wPaper;
    MoveL Offs(pOrigin,179.66,79.16,0.00),v40,z0,tPen\WObj:=wPaper;
    MoveL Offs(pOrigin,179.45,78.36,0.00),v40,z0,tPen\WObj:=wPaper;
    MoveL Offs(pOrigin,183.06,78.36,0.00),v40,fine,tPen\WObj:=wPaper;
    MoveL Offs(pOrigin,183.06,78.36,6.00),v60,z5,tPen\WObj:=wPaper;
    MoveL Offs(pOrigin,184.31,80.06,6.00),vTravel,z5,tPen\WObj:=wPaper;
    MoveL Offs(pOrigin,184.31,80.06,0.00),v60,z0,tPen\WObj:=wPaper;
    MoveL Offs(pOrigin,181.00,76.76,0.00),v40,z0,tPen\WObj:=wPaper;
    MoveL Offs(pOrigin,181.01,76.11,0.00),v40,z0,tPen\WObj:=wPaper;
    MoveL Offs(pOrigin,177.85,79.26,0.00),v40,z0,tPen\WObj:=wPaper;
    MoveL Offs(pOrigin,178.32,80.04,0.00),v40,z0,tPen\WObj:=wPaper;
  ENDPROC

  PROC DrawPart261()
    MoveL Offs(pOrigin,181.02,82.75,0.00),v40,fine,tPen\WObj:=wPaper;
    MoveL Offs(pOrigin,181.02,82.75,6.00),v60,z5,tPen\WObj:=wPaper;
    MoveL Offs(pOrigin,182.82,81.56,6.00),vTravel,z5,tPen\WObj:=wPaper;
    MoveL Offs(pOrigin,182.82,81.56,0.00),v60,z0,tPen\WObj:=wPaper;
    MoveL Offs(pOrigin,176.65,75.40,0.00),v40,z0,tPen\WObj:=wPaper;
    MoveL Offs(pOrigin,177.42,75.22,0.00),v40,z0,tPen\WObj:=wPaper;
    MoveL Offs(pOrigin,175.16,77.47,0.00),v40,z0,tPen\WObj:=wPaper;
    MoveL Offs(pOrigin,174.27,76.88,0.00),v40,z0,tPen\WObj:=wPaper;
    MoveL Offs(pOrigin,176.52,74.62,0.00),v40,z0,tPen\WObj:=wPaper;
    MoveL Offs(pOrigin,175.84,75.19,0.00),v40,z0,tPen\WObj:=wPaper;
    MoveL Offs(pOrigin,174.35,75.19,0.00),v40,z0,tPen\WObj:=wPaper;
    MoveL Offs(pOrigin,174.77,75.97,0.00),v40,z0,tPen\WObj:=wPaper;
    MoveL Offs(pOrigin,175.20,76.40,0.00),v40,z0,tPen\WObj:=wPaper;
    MoveL Offs(pOrigin,174.77,75.97,0.00),v40,fine,tPen\WObj:=wPaper;
    MoveL Offs(pOrigin,174.77,75.97,6.00),v60,z5,tPen\WObj:=wPaper;
    MoveL Offs(pOrigin,173.52,76.13,6.00),vTravel,z5,tPen\WObj:=wPaper;
    MoveL Offs(pOrigin,173.52,76.13,0.00),v60,z0,tPen\WObj:=wPaper;
    MoveL Offs(pOrigin,175.77,73.88,0.00),v40,z0,tPen\WObj:=wPaper;
    MoveL Offs(pOrigin,174.99,74.28,0.00),v40,z0,tPen\WObj:=wPaper;
    MoveL Offs(pOrigin,175.62,74.91,0.00),v40,z0,tPen\WObj:=wPaper;
    MoveL Offs(pOrigin,174.99,74.28,0.00),v40,z0,tPen\WObj:=wPaper;
    MoveL Offs(pOrigin,174.56,74.14,0.00),v40,z0,tPen\WObj:=wPaper;
    MoveL Offs(pOrigin,173.29,74.14,0.00),v40,z0,tPen\WObj:=wPaper;
    MoveL Offs(pOrigin,173.07,74.49,0.00),v40,z0,tPen\WObj:=wPaper;
    MoveL Offs(pOrigin,173.50,74.91,0.00),v40,z0,tPen\WObj:=wPaper;
    MoveL Offs(pOrigin,173.07,74.49,0.00),v40,z0,tPen\WObj:=wPaper;
    MoveL Offs(pOrigin,172.77,75.38,0.00),v40,z0,tPen\WObj:=wPaper;
    MoveL Offs(pOrigin,174.88,73.28,0.00),v40,z0,tPen\WObj:=wPaper;
    MoveL Offs(pOrigin,173.93,73.21,0.00),v40,z0,tPen\WObj:=wPaper;
    MoveL Offs(pOrigin,174.77,74.06,0.00),v40,z0,tPen\WObj:=wPaper;
    MoveL Offs(pOrigin,173.93,73.21,0.00),v40,z0,tPen\WObj:=wPaper;
    MoveL Offs(pOrigin,173.50,73.08,0.00),v40,z0,tPen\WObj:=wPaper;
    MoveL Offs(pOrigin,161.39,73.08,0.00),v40,fine,tPen\WObj:=wPaper;
    MoveL Offs(pOrigin,161.39,73.08,6.00),v60,z5,tPen\WObj:=wPaper;
    MoveL Offs(pOrigin,164.79,72.02,6.00),vTravel,z5,tPen\WObj:=wPaper;
    MoveL Offs(pOrigin,164.79,72.02,0.00),v60,z0,tPen\WObj:=wPaper;
    MoveL Offs(pOrigin,166.70,72.02,0.00),v40,fine,tPen\WObj:=wPaper;
    MoveL Offs(pOrigin,166.70,72.02,6.00),v60,z5,tPen\WObj:=wPaper;
    MoveL Offs(pOrigin,165.64,71.30,6.00),vTravel,z5,tPen\WObj:=wPaper;
    MoveL Offs(pOrigin,165.64,71.30,0.00),v60,z0,tPen\WObj:=wPaper;
    MoveL Offs(pOrigin,163.94,72.22,0.00),v40,z0,tPen\WObj:=wPaper;
    MoveL Offs(pOrigin,160.11,73.43,0.00),v40,z0,tPen\WObj:=wPaper;
    MoveL Offs(pOrigin,157.35,73.85,0.00),v40,z0,tPen\WObj:=wPaper;
    MoveL Offs(pOrigin,151.61,73.64,0.00),v40,z0,tPen\WObj:=wPaper;
    MoveL Offs(pOrigin,147.15,72.57,0.00),v40,z0,tPen\WObj:=wPaper;
    MoveL Offs(pOrigin,138.23,69.25,0.00),v40,z0,tPen\WObj:=wPaper;
    MoveL Offs(pOrigin,133.76,66.55,0.00),v40,z0,tPen\WObj:=wPaper;
    MoveL Offs(pOrigin,131.64,64.85,0.00),v40,z0,tPen\WObj:=wPaper;
    MoveL Offs(pOrigin,130.15,64.29,0.00),v40,z0,tPen\WObj:=wPaper;
    MoveL Offs(pOrigin,129.90,64.50,0.00),v40,z0,tPen\WObj:=wPaper;
    MoveL Offs(pOrigin,129.90,65.99,0.00),v40,fine,tPen\WObj:=wPaper;
    MoveL Offs(pOrigin,129.90,65.99,6.00),v60,z5,tPen\WObj:=wPaper;
    MoveL Offs(pOrigin,128.66,65.69,6.00),vTravel,z5,tPen\WObj:=wPaper;
    MoveL Offs(pOrigin,128.66,65.69,0.00),v60,z0,tPen\WObj:=wPaper;
    MoveL Offs(pOrigin,132.70,65.69,0.00),v40,z0,tPen\WObj:=wPaper;
    MoveL Offs(pOrigin,132.01,65.78,0.00),v40,z0,tPen\WObj:=wPaper;
    MoveL Offs(pOrigin,132.01,67.26,0.00),v40,fine,tPen\WObj:=wPaper;
    MoveL Offs(pOrigin,132.01,67.26,6.00),v60,z5,tPen\WObj:=wPaper;
    MoveL Offs(pOrigin,133.07,66.62,6.00),vTravel,z5,tPen\WObj:=wPaper;
    MoveL Offs(pOrigin,133.07,66.62,0.00),v60,z0,tPen\WObj:=wPaper;
    MoveL Offs(pOrigin,133.07,67.90,0.00),v40,fine,tPen\WObj:=wPaper;
    MoveL Offs(pOrigin,133.07,67.90,6.00),v60,z5,tPen\WObj:=wPaper;
    MoveL Offs(pOrigin,130.85,68.02,6.00),vTravel,z5,tPen\WObj:=wPaper;
    MoveL Offs(pOrigin,130.85,68.02,0.00),v60,z0,tPen\WObj:=wPaper;
    MoveL Offs(pOrigin,133.71,65.17,0.00),v40,z0,tPen\WObj:=wPaper;
    MoveL Offs(pOrigin,132.81,64.57,0.00),v40,z0,tPen\WObj:=wPaper;
    MoveL Offs(pOrigin,129.80,67.58,0.00),v40,fine,tPen\WObj:=wPaper;
    MoveL Offs(pOrigin,129.80,67.58,6.00),v60,z5,tPen\WObj:=wPaper;
    MoveL Offs(pOrigin,132.06,64.93,6.00),vTravel,z5,tPen\WObj:=wPaper;
    MoveL Offs(pOrigin,132.06,64.93,0.00),v60,z0,tPen\WObj:=wPaper;
    MoveL Offs(pOrigin,132.91,65.78,0.00),v40,z0,tPen\WObj:=wPaper;
    MoveL Offs(pOrigin,132.06,64.93,0.00),v40,fine,tPen\WObj:=wPaper;
    MoveL Offs(pOrigin,132.06,64.93,6.00),v60,z5,tPen\WObj:=wPaper;
    MoveL Offs(pOrigin,129.94,63.58,6.00),vTravel,z5,tPen\WObj:=wPaper;
    MoveL Offs(pOrigin,129.94,63.58,0.00),v60,z0,tPen\WObj:=wPaper;
    MoveL Offs(pOrigin,125.48,63.58,0.00),v40,z0,tPen\WObj:=wPaper;
    MoveL Offs(pOrigin,125.32,64.59,0.00),v40,z0,tPen\WObj:=wPaper;
    MoveL Offs(pOrigin,129.23,60.69,0.00),v40,z0,tPen\WObj:=wPaper;
    MoveL Offs(pOrigin,128.48,59.94,0.00),v40,z0,tPen\WObj:=wPaper;
    MoveL Offs(pOrigin,124.42,64.00,0.00),v40,z0,tPen\WObj:=wPaper;
    MoveL Offs(pOrigin,123.52,63.40,0.00),v40,z0,tPen\WObj:=wPaper;
    MoveL Offs(pOrigin,127.88,59.04,0.00),v40,z0,tPen\WObj:=wPaper;
    MoveL Offs(pOrigin,127.44,58.00,0.00),v40,z0,tPen\WObj:=wPaper;
    MoveL Offs(pOrigin,122.78,62.65,0.00),v40,z0,tPen\WObj:=wPaper;
    MoveL Offs(pOrigin,123.78,62.38,0.00),v40,z0,tPen\WObj:=wPaper;
    MoveL Offs(pOrigin,124.41,63.01,0.00),v40,z0,tPen\WObj:=wPaper;
    MoveL Offs(pOrigin,123.78,62.38,0.00),v40,z0,tPen\WObj:=wPaper;
    MoveL Offs(pOrigin,124.20,62.52,0.00),v40,z0,tPen\WObj:=wPaper;
    MoveL Offs(pOrigin,126.32,62.52,0.00),v40,fine,tPen\WObj:=wPaper;
    MoveL Offs(pOrigin,126.32,62.52,6.00),v60,z5,tPen\WObj:=wPaper;
    MoveL Offs(pOrigin,127.81,61.95,6.00),vTravel,z5,tPen\WObj:=wPaper;
    MoveL Offs(pOrigin,127.81,61.95,0.00),v60,z0,tPen\WObj:=wPaper;
    MoveL Offs(pOrigin,128.24,62.59,0.00),v40,z0,tPen\WObj:=wPaper;
    MoveL Offs(pOrigin,127.81,61.95,0.00),v40,fine,tPen\WObj:=wPaper;
    MoveL Offs(pOrigin,127.81,61.95,6.00),v60,z5,tPen\WObj:=wPaper;
    MoveL Offs(pOrigin,128.45,63.65,6.00),vTravel,z5,tPen\WObj:=wPaper;
    MoveL Offs(pOrigin,128.45,63.65,0.00),v60,z0,tPen\WObj:=wPaper;
    MoveL Offs(pOrigin,126.96,63.01,0.00),v40,z0,tPen\WObj:=wPaper;
    MoveL Offs(pOrigin,123.78,60.04,0.00),v40,z0,tPen\WObj:=wPaper;
    MoveL Offs(pOrigin,122.07,56.42,0.00),v40,z0,tPen\WObj:=wPaper;
    MoveL Offs(pOrigin,121.86,55.36,0.00),v40,z0,tPen\WObj:=wPaper;
    MoveL Offs(pOrigin,122.29,54.72,0.00),v40,z0,tPen\WObj:=wPaper;
    MoveL Offs(pOrigin,122.29,55.13,0.00),v40,z0,tPen\WObj:=wPaper;
    MoveL Offs(pOrigin,120.38,55.13,0.00),v40,z0,tPen\WObj:=wPaper;
    MoveL Offs(pOrigin,120.40,54.51,0.00),v40,z0,tPen\WObj:=wPaper;
    MoveL Offs(pOrigin,120.40,48.56,0.00),v40,z0,tPen\WObj:=wPaper;
    MoveL Offs(pOrigin,121.01,48.79,0.00),v40,z0,tPen\WObj:=wPaper;
    MoveL Offs(pOrigin,119.52,48.79,0.00),v40,z0,tPen\WObj:=wPaper;
    MoveL Offs(pOrigin,118.63,48.89,0.00),v40,z0,tPen\WObj:=wPaper;
    MoveL Offs(pOrigin,131.10,36.41,0.00),v40,z0,tPen\WObj:=wPaper;
    MoveL Offs(pOrigin,131.00,37.18,0.00),v40,z0,tPen\WObj:=wPaper;
    MoveL Offs(pOrigin,145.02,37.18,0.00),v40,fine,tPen\WObj:=wPaper;
    MoveL Offs(pOrigin,145.02,37.18,6.00),v60,z5,tPen\WObj:=wPaper;
    MoveL Offs(pOrigin,144.33,35.60,6.00),vTravel,z5,tPen\WObj:=wPaper;
    MoveL Offs(pOrigin,144.33,35.60,0.00),v60,z0,tPen\WObj:=wPaper;
    MoveL Offs(pOrigin,150.19,41.46,0.00),v40,z0,tPen\WObj:=wPaper;
    MoveL Offs(pOrigin,149.97,40.49,0.00),v40,z0,tPen\WObj:=wPaper;
    MoveL Offs(pOrigin,149.97,38.79,0.00),v40,z0,tPen\WObj:=wPaper;
    MoveL Offs(pOrigin,148.91,38.79,0.00),v40,z0,tPen\WObj:=wPaper;
    MoveL Offs(pOrigin,148.91,40.70,0.00),v40,z0,tPen\WObj:=wPaper;
  ENDPROC

  PROC DrawPart262()
    MoveL Offs(pOrigin,149.06,39.85,0.00),v40,z0,tPen\WObj:=wPaper;
    MoveL Offs(pOrigin,146.09,40.49,0.00),v40,z0,tPen\WObj:=wPaper;
    MoveL Offs(pOrigin,144.39,41.27,0.00),v40,z0,tPen\WObj:=wPaper;
    MoveL Offs(pOrigin,143.75,42.26,0.00),v40,z0,tPen\WObj:=wPaper;
    MoveL Offs(pOrigin,142.76,42.83,0.00),v40,z0,tPen\WObj:=wPaper;
    MoveL Offs(pOrigin,141.84,44.31,0.00),v40,z0,tPen\WObj:=wPaper;
    MoveL Offs(pOrigin,141.84,44.31,0.00),v40,z0,tPen\WObj:=wPaper;
    MoveL Offs(pOrigin,141.77,45.38,0.00),v40,z0,tPen\WObj:=wPaper;
    MoveL Offs(pOrigin,141.20,46.22,0.00),v40,z0,tPen\WObj:=wPaper;
    MoveL Offs(pOrigin,141.41,46.86,0.00),v40,z0,tPen\WObj:=wPaper;
    MoveL Offs(pOrigin,141.20,47.92,0.00),v40,z0,tPen\WObj:=wPaper;
    MoveL Offs(pOrigin,141.20,47.92,0.00),v40,z0,tPen\WObj:=wPaper;
    MoveL Offs(pOrigin,141.62,48.35,0.00),v40,z0,tPen\WObj:=wPaper;
    MoveL Offs(pOrigin,141.62,50.26,0.00),v40,z0,tPen\WObj:=wPaper;
    MoveL Offs(pOrigin,142.57,49.62,0.00),v40,z0,tPen\WObj:=wPaper;
    MoveL Offs(pOrigin,142.57,54.51,0.00),v40,z0,tPen\WObj:=wPaper;
    MoveL Offs(pOrigin,142.48,53.66,0.00),v40,z0,tPen\WObj:=wPaper;
    MoveL Offs(pOrigin,145.45,60.46,0.00),v40,z0,tPen\WObj:=wPaper;
    MoveL Offs(pOrigin,145.24,61.31,0.00),v40,z0,tPen\WObj:=wPaper;
    MoveL Offs(pOrigin,145.74,60.68,0.00),v40,z0,tPen\WObj:=wPaper;
    MoveL Offs(pOrigin,145.74,58.76,0.00),v40,z0,tPen\WObj:=wPaper;
    MoveL Offs(pOrigin,146.30,58.30,0.00),v40,z0,tPen\WObj:=wPaper;
    MoveL Offs(pOrigin,140.35,58.30,0.00),v40,z0,tPen\WObj:=wPaper;
    MoveL Offs(pOrigin,140.35,58.34,0.00),v40,z0,tPen\WObj:=wPaper;
    MoveL Offs(pOrigin,140.56,58.76,0.00),v40,z0,tPen\WObj:=wPaper;
    MoveL Offs(pOrigin,140.35,58.34,0.00),v40,z0,tPen\WObj:=wPaper;
    MoveL Offs(pOrigin,140.46,57.28,0.00),v40,z0,tPen\WObj:=wPaper;
    MoveL Offs(pOrigin,140.46,56.21,0.00),v40,z0,tPen\WObj:=wPaper;
    MoveL Offs(pOrigin,139.93,57.24,0.00),v40,z0,tPen\WObj:=wPaper;
    MoveL Offs(pOrigin,145.45,57.24,0.00),v40,z0,tPen\WObj:=wPaper;
    MoveL Offs(pOrigin,145.45,56.85,0.00),v40,z0,tPen\WObj:=wPaper;
    MoveL Offs(pOrigin,145.66,57.28,0.00),v40,z0,tPen\WObj:=wPaper;
    MoveL Offs(pOrigin,145.45,56.85,0.00),v40,z0,tPen\WObj:=wPaper;
    MoveL Offs(pOrigin,145.02,56.18,0.00),v40,z0,tPen\WObj:=wPaper;
    MoveL Offs(pOrigin,139.29,56.18,0.00),v40,z0,tPen\WObj:=wPaper;
    MoveL Offs(pOrigin,139.07,55.13,0.00),v40,z0,tPen\WObj:=wPaper;
    MoveL Offs(pOrigin,144.60,55.13,0.00),v40,z0,tPen\WObj:=wPaper;
    MoveL Offs(pOrigin,145.14,55.83,0.00),v40,z0,tPen\WObj:=wPaper;
    MoveL Offs(pOrigin,136.72,47.41,0.00),v40,z0,tPen\WObj:=wPaper;
    MoveL Offs(pOrigin,136.95,47.50,0.00),v40,z0,tPen\WObj:=wPaper;
    MoveL Offs(pOrigin,136.74,47.92,0.00),v40,z0,tPen\WObj:=wPaper;
    MoveL Offs(pOrigin,136.95,47.50,0.00),v40,z0,tPen\WObj:=wPaper;
    MoveL Offs(pOrigin,137.16,47.74,0.00),v40,z0,tPen\WObj:=wPaper;
    MoveL Offs(pOrigin,143.11,47.74,0.00),v40,z0,tPen\WObj:=wPaper;
    MoveL Offs(pOrigin,142.57,47.08,0.00),v40,z0,tPen\WObj:=wPaper;
    MoveL Offs(pOrigin,142.57,44.31,0.00),v40,z0,tPen\WObj:=wPaper;
    MoveL Offs(pOrigin,141.84,44.31,0.00),v40,z0,tPen\WObj:=wPaper;
    MoveL Offs(pOrigin,140.99,44.74,0.00),v40,z0,tPen\WObj:=wPaper;
    MoveL Offs(pOrigin,141.20,45.80,0.00),v40,z0,tPen\WObj:=wPaper;
    MoveL Offs(pOrigin,140.46,45.80,0.00),v40,z0,tPen\WObj:=wPaper;
    MoveL Offs(pOrigin,140.46,43.46,0.00),v40,z0,tPen\WObj:=wPaper;
    MoveL Offs(pOrigin,139.70,42.93,0.00),v40,z0,tPen\WObj:=wPaper;
    MoveL Offs(pOrigin,143.76,46.98,0.00),v40,z0,tPen\WObj:=wPaper;
    MoveL Offs(pOrigin,144.25,47.16,0.00),v40,z0,tPen\WObj:=wPaper;
    MoveL Offs(pOrigin,135.38,56.02,0.00),v40,z0,tPen\WObj:=wPaper;
    MoveL Offs(pOrigin,136.52,56.18,0.00),v40,z0,tPen\WObj:=wPaper;
    MoveL Offs(pOrigin,137.59,56.18,0.00),v40,fine,tPen\WObj:=wPaper;
    MoveL Offs(pOrigin,137.59,56.18,6.00),v60,z5,tPen\WObj:=wPaper;
    MoveL Offs(pOrigin,135.68,57.22,6.00),vTravel,z5,tPen\WObj:=wPaper;
    MoveL Offs(pOrigin,135.68,57.22,0.00),v60,z0,tPen\WObj:=wPaper;
    MoveL Offs(pOrigin,143.94,48.96,0.00),v40,z0,tPen\WObj:=wPaper;
    MoveL Offs(pOrigin,143.47,49.68,0.00),v40,z0,tPen\WObj:=wPaper;
    MoveL Offs(pOrigin,138.21,44.42,0.00),v40,fine,tPen\WObj:=wPaper;
    MoveL Offs(pOrigin,138.21,44.42,6.00),v60,z5,tPen\WObj:=wPaper;
    MoveL Offs(pOrigin,136.62,44.34,6.00),vTravel,z5,tPen\WObj:=wPaper;
    MoveL Offs(pOrigin,136.62,44.34,0.00),v60,z0,tPen\WObj:=wPaper;
    MoveL Offs(pOrigin,146.08,34.87,0.00),v40,z0,tPen\WObj:=wPaper;
    MoveL Offs(pOrigin,145.82,35.60,0.00),v40,z0,tPen\WObj:=wPaper;
    MoveL Offs(pOrigin,151.23,41.01,0.00),v40,z0,tPen\WObj:=wPaper;
    MoveL Offs(pOrigin,151.45,41.44,0.00),v40,z0,tPen\WObj:=wPaper;
    MoveL Offs(pOrigin,159.57,33.33,0.00),v40,z0,tPen\WObj:=wPaper;
    MoveL Offs(pOrigin,160.35,33.70,0.00),v40,z0,tPen\WObj:=wPaper;
    MoveL Offs(pOrigin,161.70,35.05,0.00),v40,z0,tPen\WObj:=wPaper;
    MoveL Offs(pOrigin,161.96,35.42,0.00),v40,z0,tPen\WObj:=wPaper;
    MoveL Offs(pOrigin,166.47,30.91,0.00),v40,z0,tPen\WObj:=wPaper;
    MoveL Offs(pOrigin,166.04,31.92,0.00),v40,z0,tPen\WObj:=wPaper;
    MoveL Offs(pOrigin,167.39,33.27,0.00),v40,z0,tPen\WObj:=wPaper;
    MoveL Offs(pOrigin,166.49,32.95,0.00),v40,z0,tPen\WObj:=wPaper;
    MoveL Offs(pOrigin,162.88,32.95,0.00),v40,z0,tPen\WObj:=wPaper;
    MoveL Offs(pOrigin,163.64,32.51,0.00),v40,z0,tPen\WObj:=wPaper;
    MoveL Offs(pOrigin,164.99,33.87,0.00),v40,fine,tPen\WObj:=wPaper;
    MoveL Offs(pOrigin,164.99,33.87,6.00),v60,z5,tPen\WObj:=wPaper;
    MoveL Offs(pOrigin,162.66,34.01,6.00),vTravel,z5,tPen\WObj:=wPaper;
    MoveL Offs(pOrigin,162.66,34.01,0.00),v60,z0,tPen\WObj:=wPaper;
    MoveL Offs(pOrigin,160.54,34.01,0.00),v40,z0,tPen\WObj:=wPaper;
    MoveL Offs(pOrigin,160.54,33.90,0.00),v40,z0,tPen\WObj:=wPaper;
    MoveL Offs(pOrigin,165.43,31.99,0.00),v40,z0,tPen\WObj:=wPaper;
    MoveL Offs(pOrigin,170.10,31.35,0.00),v40,z0,tPen\WObj:=wPaper;
    MoveL Offs(pOrigin,179.88,31.56,0.00),v40,z0,tPen\WObj:=wPaper;
    MoveL Offs(pOrigin,183.91,31.14,0.00),v40,z0,tPen\WObj:=wPaper;
    MoveL Offs(pOrigin,190.50,31.14,0.00),v40,z0,tPen\WObj:=wPaper;
    MoveL Offs(pOrigin,195.81,31.77,0.00),v40,z0,tPen\WObj:=wPaper;
    MoveL Offs(pOrigin,200.91,33.26,0.00),v40,z0,tPen\WObj:=wPaper;
    MoveL Offs(pOrigin,218.76,32.20,0.00),v40,fine,tPen\WObj:=wPaper;
    MoveL Offs(pOrigin,218.76,32.20,6.00),v60,z5,tPen\WObj:=wPaper;
    MoveL Offs(pOrigin,222.17,39.43,6.00),vTravel,z5,tPen\WObj:=wPaper;
    MoveL Offs(pOrigin,222.17,39.43,0.00),v60,z0,tPen\WObj:=wPaper;
    MoveL Offs(pOrigin,213.75,47.84,0.00),v40,fine,tPen\WObj:=wPaper;
    MoveL Offs(pOrigin,213.75,47.84,6.00),v60,z5,tPen\WObj:=wPaper;
    MoveL Offs(pOrigin,213.43,54.14,6.00),vTravel,z5,tPen\WObj:=wPaper;
    MoveL Offs(pOrigin,213.43,54.14,0.00),v60,z0,tPen\WObj:=wPaper;
    MoveL Offs(pOrigin,228.61,38.96,0.00),v40,fine,tPen\WObj:=wPaper;
    MoveL Offs(pOrigin,228.61,38.96,6.00),v60,z5,tPen\WObj:=wPaper;
    MoveL Offs(pOrigin,226.62,43.04,6.00),vTravel,z5,tPen\WObj:=wPaper;
    MoveL Offs(pOrigin,226.62,43.04,0.00),v60,z0,tPen\WObj:=wPaper;
    MoveL Offs(pOrigin,226.20,43.67,0.00),v40,z0,tPen\WObj:=wPaper;
    MoveL Offs(pOrigin,226.62,43.04,0.00),v40,fine,tPen\WObj:=wPaper;
    MoveL Offs(pOrigin,226.62,43.04,6.00),v60,z5,tPen\WObj:=wPaper;
    MoveL Offs(pOrigin,224.71,45.62,6.00),vTravel,z5,tPen\WObj:=wPaper;
    MoveL Offs(pOrigin,224.71,45.62,0.00),v60,z0,tPen\WObj:=wPaper;
    MoveL Offs(pOrigin,223.44,45.62,0.00),v40,fine,tPen\WObj:=wPaper;
    MoveL Offs(pOrigin,223.44,45.62,6.00),v60,z5,tPen\WObj:=wPaper;
    MoveL Offs(pOrigin,224.50,46.22,6.00),vTravel,z5,tPen\WObj:=wPaper;
    MoveL Offs(pOrigin,224.50,46.22,0.00),v60,z0,tPen\WObj:=wPaper;
    MoveL Offs(pOrigin,224.07,46.86,0.00),v40,z0,tPen\WObj:=wPaper;
    MoveL Offs(pOrigin,224.50,46.22,0.00),v40,fine,tPen\WObj:=wPaper;
    MoveL Offs(pOrigin,224.50,46.22,6.00),v60,z5,tPen\WObj:=wPaper;
    MoveL Offs(pOrigin,222.80,48.56,6.00),vTravel,z5,tPen\WObj:=wPaper;
    MoveL Offs(pOrigin,222.80,48.56,0.00),v60,z0,tPen\WObj:=wPaper;
    MoveL Offs(pOrigin,222.38,49.20,0.00),v40,z0,tPen\WObj:=wPaper;
  ENDPROC

  PROC DrawPart263()
    MoveL Offs(pOrigin,222.80,48.56,0.00),v40,fine,tPen\WObj:=wPaper;
    MoveL Offs(pOrigin,222.80,48.56,6.00),v60,z5,tPen\WObj:=wPaper;
    MoveL Offs(pOrigin,217.55,42.40,6.00),vTravel,z5,tPen\WObj:=wPaper;
    MoveL Offs(pOrigin,217.55,42.40,0.00),v60,z0,tPen\WObj:=wPaper;
    MoveL Offs(pOrigin,217.55,41.12,0.00),v40,fine,tPen\WObj:=wPaper;
    MoveL Offs(pOrigin,217.55,41.12,6.00),v60,z5,tPen\WObj:=wPaper;
    MoveL Offs(pOrigin,203.23,45.22,6.00),vTravel,z5,tPen\WObj:=wPaper;
    MoveL Offs(pOrigin,203.23,45.22,0.00),v60,z0,tPen\WObj:=wPaper;
    MoveL Offs(pOrigin,201.72,43.72,0.00),v40,fine,tPen\WObj:=wPaper;
    MoveL Offs(pOrigin,201.72,43.72,6.00),v60,z5,tPen\WObj:=wPaper;
    MoveL Offs(pOrigin,203.04,44.57,6.00),vTravel,z5,tPen\WObj:=wPaper;
    MoveL Offs(pOrigin,203.04,44.57,0.00),v60,z0,tPen\WObj:=wPaper;
    MoveL Offs(pOrigin,199.64,44.57,0.00),v40,z0,tPen\WObj:=wPaper;
    MoveL Offs(pOrigin,199.33,44.31,0.00),v40,z0,tPen\WObj:=wPaper;
    MoveL Offs(pOrigin,200.83,45.81,0.00),v40,fine,tPen\WObj:=wPaper;
    MoveL Offs(pOrigin,200.83,45.81,6.00),v60,z5,tPen\WObj:=wPaper;
    MoveL Offs(pOrigin,199.00,45.62,6.00),vTravel,z5,tPen\WObj:=wPaper;
    MoveL Offs(pOrigin,199.00,45.62,0.00),v60,z0,tPen\WObj:=wPaper;
    MoveL Offs(pOrigin,196.02,45.62,0.00),v40,z0,tPen\WObj:=wPaper;
    MoveL Offs(pOrigin,195.89,45.35,0.00),v40,z0,tPen\WObj:=wPaper;
    MoveL Offs(pOrigin,197.24,46.70,0.00),v40,fine,tPen\WObj:=wPaper;
    MoveL Offs(pOrigin,197.24,46.70,6.00),v60,z5,tPen\WObj:=wPaper;
    MoveL Offs(pOrigin,190.50,48.92,6.00),vTravel,z5,tPen\WObj:=wPaper;
    MoveL Offs(pOrigin,190.50,48.92,0.00),v60,z0,tPen\WObj:=wPaper;
    MoveL Offs(pOrigin,184.34,42.76,0.00),v40,fine,tPen\WObj:=wPaper;
    MoveL Offs(pOrigin,184.34,42.76,6.00),v60,z5,tPen\WObj:=wPaper;
    MoveL Offs(pOrigin,181.41,41.35,6.00),vTravel,z5,tPen\WObj:=wPaper;
    MoveL Offs(pOrigin,181.41,41.35,0.00),v60,z0,tPen\WObj:=wPaper;
    MoveL Offs(pOrigin,185.77,36.99,0.00),v40,fine,tPen\WObj:=wPaper;
    MoveL Offs(pOrigin,185.77,36.99,6.00),v60,z5,tPen\WObj:=wPaper;
    MoveL Offs(pOrigin,192.56,36.05,6.00),vTravel,z5,tPen\WObj:=wPaper;
    MoveL Offs(pOrigin,192.56,36.05,0.00),v60,z0,tPen\WObj:=wPaper;
    MoveL Offs(pOrigin,193.91,37.40,0.00),v40,fine,tPen\WObj:=wPaper;
    MoveL Offs(pOrigin,193.91,37.40,6.00),v60,z5,tPen\WObj:=wPaper;
    MoveL Offs(pOrigin,196.90,24.38,6.00),vTravel,z5,tPen\WObj:=wPaper;
    MoveL Offs(pOrigin,196.90,24.38,0.00),v60,z0,tPen\WObj:=wPaper;
    MoveL Offs(pOrigin,200.50,20.77,0.00),v40,fine,tPen\WObj:=wPaper;
    MoveL Offs(pOrigin,200.50,20.77,6.00),v60,z5,tPen\WObj:=wPaper;
    MoveL Offs(pOrigin,199.00,20.78,6.00),vTravel,z5,tPen\WObj:=wPaper;
    MoveL Offs(pOrigin,199.00,20.78,0.00),v60,z0,tPen\WObj:=wPaper;
    MoveL Offs(pOrigin,195.85,23.93,0.00),v40,z0,tPen\WObj:=wPaper;
    MoveL Offs(pOrigin,196.72,23.78,0.00),v40,z0,tPen\WObj:=wPaper;
    MoveL Offs(pOrigin,188.61,15.66,0.00),v40,z0,tPen\WObj:=wPaper;
    MoveL Offs(pOrigin,188.24,15.12,0.00),v40,z0,tPen\WObj:=wPaper;
    MoveL Offs(pOrigin,178.77,24.58,0.00),v40,fine,tPen\WObj:=wPaper;
    MoveL Offs(pOrigin,178.77,24.58,6.00),v60,z5,tPen\WObj:=wPaper;
    MoveL Offs(pOrigin,180.27,24.58,6.00),vTravel,z5,tPen\WObj:=wPaper;
    MoveL Offs(pOrigin,180.27,24.58,0.00),v60,z0,tPen\WObj:=wPaper;
    MoveL Offs(pOrigin,189.88,14.96,0.00),v40,fine,tPen\WObj:=wPaper;
    MoveL Offs(pOrigin,189.88,14.96,6.00),v60,z5,tPen\WObj:=wPaper;
    MoveL Offs(pOrigin,187.41,15.96,6.00),vTravel,z5,tPen\WObj:=wPaper;
    MoveL Offs(pOrigin,187.41,15.96,0.00),v60,z0,tPen\WObj:=wPaper;
    MoveL Offs(pOrigin,191.61,20.17,0.00),v40,fine,tPen\WObj:=wPaper;
    MoveL Offs(pOrigin,191.61,20.17,6.00),v60,z5,tPen\WObj:=wPaper;
    MoveL Offs(pOrigin,190.12,20.16,6.00),vTravel,z5,tPen\WObj:=wPaper;
    MoveL Offs(pOrigin,190.12,20.16,0.00),v60,z0,tPen\WObj:=wPaper;
    MoveL Offs(pOrigin,186.06,16.10,0.00),v40,fine,tPen\WObj:=wPaper;
    MoveL Offs(pOrigin,186.06,16.10,6.00),v60,z5,tPen\WObj:=wPaper;
    MoveL Offs(pOrigin,184.94,15.43,6.00),vTravel,z5,tPen\WObj:=wPaper;
    MoveL Offs(pOrigin,184.94,15.43,0.00),v60,z0,tPen\WObj:=wPaper;
    MoveL Offs(pOrigin,175.47,24.89,0.00),v40,z0,tPen\WObj:=wPaper;
    MoveL Offs(pOrigin,175.00,24.46,0.00),v40,z0,tPen\WObj:=wPaper;
    MoveL Offs(pOrigin,173.95,23.41,0.00),v40,fine,tPen\WObj:=wPaper;
    MoveL Offs(pOrigin,173.95,23.41,6.00),v60,z5,tPen\WObj:=wPaper;
    MoveL Offs(pOrigin,175.30,23.26,6.00),vTravel,z5,tPen\WObj:=wPaper;
    MoveL Offs(pOrigin,175.30,23.26,0.00),v60,z0,tPen\WObj:=wPaper;
    MoveL Offs(pOrigin,176.20,24.16,0.00),v40,fine,tPen\WObj:=wPaper;
    MoveL Offs(pOrigin,176.20,24.16,6.00),v60,z5,tPen\WObj:=wPaper;
    MoveL Offs(pOrigin,182.00,18.17,6.00),vTravel,z5,tPen\WObj:=wPaper;
    MoveL Offs(pOrigin,182.00,18.17,0.00),v60,z0,tPen\WObj:=wPaper;
    MoveL Offs(pOrigin,168.61,18.17,0.00),v40,fine,tPen\WObj:=wPaper;
    MoveL Offs(pOrigin,168.61,18.17,6.00),v60,z5,tPen\WObj:=wPaper;
    MoveL Offs(pOrigin,184.56,16.10,6.00),vTravel,z5,tPen\WObj:=wPaper;
    MoveL Offs(pOrigin,184.56,16.10,0.00),v60,z0,tPen\WObj:=wPaper;
    MoveL Offs(pOrigin,188.92,20.46,0.00),v40,fine,tPen\WObj:=wPaper;
    MoveL Offs(pOrigin,188.92,20.46,6.00),v60,z5,tPen\WObj:=wPaper;
    MoveL Offs(pOrigin,186.46,19.22,6.00),vTravel,z5,tPen\WObj:=wPaper;
    MoveL Offs(pOrigin,186.46,19.22,0.00),v60,z0,tPen\WObj:=wPaper;
    MoveL Offs(pOrigin,194.96,19.22,0.00),v40,z0,tPen\WObj:=wPaper;
    MoveL Offs(pOrigin,194.96,18.17,0.00),v40,z0,tPen\WObj:=wPaper;
    MoveL Offs(pOrigin,192.41,18.17,0.00),v40,fine,tPen\WObj:=wPaper;
    MoveL Offs(pOrigin,192.41,18.17,6.00),v60,z5,tPen\WObj:=wPaper;
    MoveL Offs(pOrigin,199.11,21.69,6.00),vTravel,z5,tPen\WObj:=wPaper;
    MoveL Offs(pOrigin,199.11,21.69,0.00),v60,z0,tPen\WObj:=wPaper;
    MoveL Offs(pOrigin,201.06,23.64,0.00),v40,fine,tPen\WObj:=wPaper;
    MoveL Offs(pOrigin,201.06,23.64,6.00),v60,z5,tPen\WObj:=wPaper;
    MoveL Offs(pOrigin,202.24,15.85,6.00),vTravel,z5,tPen\WObj:=wPaper;
    MoveL Offs(pOrigin,202.24,15.85,0.00),v60,z0,tPen\WObj:=wPaper;
    MoveL Offs(pOrigin,200.13,13.75,0.00),v40,fine,tPen\WObj:=wPaper;
    MoveL Offs(pOrigin,200.13,13.75,6.00),v60,z5,tPen\WObj:=wPaper;
    MoveL Offs(pOrigin,206.54,53.56,6.00),vTravel,z5,tPen\WObj:=wPaper;
    MoveL Offs(pOrigin,206.54,53.56,0.00),v60,z0,tPen\WObj:=wPaper;
    MoveL Offs(pOrigin,199.78,60.32,0.00),v40,z0,tPen\WObj:=wPaper;
    MoveL Offs(pOrigin,199.83,59.74,0.00),v40,z0,tPen\WObj:=wPaper;
    MoveL Offs(pOrigin,198.47,58.39,0.00),v40,z0,tPen\WObj:=wPaper;
    MoveL Offs(pOrigin,199.64,58.30,0.00),v40,z0,tPen\WObj:=wPaper;
    MoveL Offs(pOrigin,201.55,58.30,0.00),v40,fine,tPen\WObj:=wPaper;
    MoveL Offs(pOrigin,201.55,58.30,6.00),v60,z5,tPen\WObj:=wPaper;
    MoveL Offs(pOrigin,200.87,59.29,6.00),vTravel,z5,tPen\WObj:=wPaper;
    MoveL Offs(pOrigin,200.87,59.29,0.00),v60,z0,tPen\WObj:=wPaper;
    MoveL Offs(pOrigin,199.67,58.09,0.00),v40,fine,tPen\WObj:=wPaper;
    MoveL Offs(pOrigin,199.67,58.09,6.00),v60,z5,tPen\WObj:=wPaper;
    MoveL Offs(pOrigin,201.61,57.05,6.00),vTravel,z5,tPen\WObj:=wPaper;
    MoveL Offs(pOrigin,201.61,57.05,0.00),v60,z0,tPen\WObj:=wPaper;
    MoveL Offs(pOrigin,202.97,58.40,0.00),v40,z0,tPen\WObj:=wPaper;
    MoveL Offs(pOrigin,203.86,57.80,0.00),v40,z0,tPen\WObj:=wPaper;
    MoveL Offs(pOrigin,202.51,56.45,0.00),v40,z0,tPen\WObj:=wPaper;
    MoveL Offs(pOrigin,202.19,57.24,0.00),v40,z0,tPen\WObj:=wPaper;
    MoveL Offs(pOrigin,204.10,57.24,0.00),v40,z0,tPen\WObj:=wPaper;
    MoveL Offs(pOrigin,204.31,56.18,0.00),v40,z0,tPen\WObj:=wPaper;
    MoveL Offs(pOrigin,206.01,56.18,0.00),v40,z0,tPen\WObj:=wPaper;
    MoveL Offs(pOrigin,205.96,56.91,0.00),v40,z0,tPen\WObj:=wPaper;
    MoveL Offs(pOrigin,204.61,55.56,0.00),v40,z0,tPen\WObj:=wPaper;
    MoveL Offs(pOrigin,205.50,54.96,0.00),v40,z0,tPen\WObj:=wPaper;
    MoveL Offs(pOrigin,206.86,56.31,0.00),v40,z0,tPen\WObj:=wPaper;
    MoveL Offs(pOrigin,207.90,55.87,0.00),v40,z0,tPen\WObj:=wPaper;
    MoveL Offs(pOrigin,206.55,54.52,0.00),v40,z0,tPen\WObj:=wPaper;
    MoveL Offs(pOrigin,206.23,55.13,0.00),v40,z0,tPen\WObj:=wPaper;
    MoveL Offs(pOrigin,207.92,55.13,0.00),v40,fine,tPen\WObj:=wPaper;
    MoveL Offs(pOrigin,207.92,55.13,6.00),v60,z5,tPen\WObj:=wPaper;
  ENDPROC

  PROC DrawPart264()
    MoveL Offs(pOrigin,195.59,58.54,6.00),vTravel,z5,tPen\WObj:=wPaper;
    MoveL Offs(pOrigin,195.59,58.54,0.00),v60,z0,tPen\WObj:=wPaper;
    MoveL Offs(pOrigin,191.24,62.89,0.00),v40,z0,tPen\WObj:=wPaper;
    MoveL Offs(pOrigin,191.74,62.11,0.00),v40,z0,tPen\WObj:=wPaper;
    MoveL Offs(pOrigin,190.39,60.76,0.00),v40,z0,tPen\WObj:=wPaper;
    MoveL Offs(pOrigin,189.34,61.20,0.00),v40,z0,tPen\WObj:=wPaper;
    MoveL Offs(pOrigin,190.40,62.26,0.00),v40,z0,tPen\WObj:=wPaper;
    MoveL Offs(pOrigin,189.35,62.70,0.00),v40,z0,tPen\WObj:=wPaper;
    MoveL Offs(pOrigin,188.30,61.65,0.00),v40,fine,tPen\WObj:=wPaper;
    MoveL Offs(pOrigin,188.30,61.65,6.00),v60,z5,tPen\WObj:=wPaper;
    MoveL Offs(pOrigin,187.20,60.96,6.00),vTravel,z5,tPen\WObj:=wPaper;
    MoveL Offs(pOrigin,187.20,60.96,0.00),v60,z0,tPen\WObj:=wPaper;
    MoveL Offs(pOrigin,183.14,65.02,0.00),v40,z0,tPen\WObj:=wPaper;
    MoveL Offs(pOrigin,182.39,64.27,0.00),v40,z0,tPen\WObj:=wPaper;
    MoveL Offs(pOrigin,184.95,61.71,0.00),v40,z0,tPen\WObj:=wPaper;
    MoveL Offs(pOrigin,185.00,62.84,0.00),v40,z0,tPen\WObj:=wPaper;
    MoveL Offs(pOrigin,185.91,63.74,0.00),v40,z0,tPen\WObj:=wPaper;
    MoveL Offs(pOrigin,185.09,64.56,0.00),v40,z0,tPen\WObj:=wPaper;
    MoveL Offs(pOrigin,189.30,60.35,0.00),v40,fine,tPen\WObj:=wPaper;
    MoveL Offs(pOrigin,189.30,60.35,6.00),v60,z5,tPen\WObj:=wPaper;
    MoveL Offs(pOrigin,192.79,60.17,6.00),vTravel,z5,tPen\WObj:=wPaper;
    MoveL Offs(pOrigin,192.79,60.17,0.00),v60,z0,tPen\WObj:=wPaper;
    MoveL Offs(pOrigin,194.14,61.52,0.00),v40,fine,tPen\WObj:=wPaper;
    MoveL Offs(pOrigin,194.14,61.52,6.00),v60,z5,tPen\WObj:=wPaper;
    MoveL Offs(pOrigin,193.48,60.41,6.00),vTravel,z5,tPen\WObj:=wPaper;
    MoveL Offs(pOrigin,193.48,60.41,0.00),v60,z0,tPen\WObj:=wPaper;
    MoveL Offs(pOrigin,195.60,60.41,0.00),v40,z0,tPen\WObj:=wPaper;
    MoveL Offs(pOrigin,196.38,60.78,0.00),v40,z0,tPen\WObj:=wPaper;
    MoveL Offs(pOrigin,195.03,59.42,0.00),v40,fine,tPen\WObj:=wPaper;
    MoveL Offs(pOrigin,195.03,59.42,6.00),v60,z5,tPen\WObj:=wPaper;
    MoveL Offs(pOrigin,184.34,63.86,6.00),vTravel,z5,tPen\WObj:=wPaper;
    MoveL Offs(pOrigin,184.34,63.86,0.00),v60,z0,tPen\WObj:=wPaper;
    MoveL Offs(pOrigin,182.85,64.71,0.00),v40,z0,tPen\WObj:=wPaper;
    MoveL Offs(pOrigin,181.57,66.20,0.00),v40,fine,tPen\WObj:=wPaper;
    MoveL Offs(pOrigin,181.57,66.20,6.00),v60,z5,tPen\WObj:=wPaper;
    MoveL Offs(pOrigin,183.91,64.07,6.00),vTravel,z5,tPen\WObj:=wPaper;
    MoveL Offs(pOrigin,183.91,64.07,0.00),v60,z0,tPen\WObj:=wPaper;
    MoveL Offs(pOrigin,184.34,63.86,0.00),v40,z0,tPen\WObj:=wPaper;
    MoveL Offs(pOrigin,183.91,64.07,0.00),v40,fine,tPen\WObj:=wPaper;
    MoveL Offs(pOrigin,183.91,64.07,6.00),v60,z5,tPen\WObj:=wPaper;
    MoveL Offs(pOrigin,189.25,73.83,6.00),vTravel,z5,tPen\WObj:=wPaper;
    MoveL Offs(pOrigin,189.25,73.83,0.00),v60,z0,tPen\WObj:=wPaper;
    MoveL Offs(pOrigin,155.00,108.09,0.00),v40,fine,tPen\WObj:=wPaper;
    MoveL Offs(pOrigin,155.00,108.09,6.00),v60,z5,tPen\WObj:=wPaper;
    MoveL Offs(pOrigin,155.14,109.44,6.00),vTravel,z5,tPen\WObj:=wPaper;
    MoveL Offs(pOrigin,155.14,109.44,0.00),v60,z0,tPen\WObj:=wPaper;
    MoveL Offs(pOrigin,152.14,112.45,0.00),v40,z0,tPen\WObj:=wPaper;
    MoveL Offs(pOrigin,152.35,112.32,0.00),v40,z0,tPen\WObj:=wPaper;
    MoveL Offs(pOrigin,150.70,110.67,0.00),v40,z0,tPen\WObj:=wPaper;
    MoveL Offs(pOrigin,150.76,111.10,0.00),v40,z0,tPen\WObj:=wPaper;
    MoveL Offs(pOrigin,153.74,111.10,0.00),v40,fine,tPen\WObj:=wPaper;
    MoveL Offs(pOrigin,153.74,111.10,6.00),v60,z5,tPen\WObj:=wPaper;
    MoveL Offs(pOrigin,154.74,110.23,6.00),vTravel,z5,tPen\WObj:=wPaper;
    MoveL Offs(pOrigin,154.74,110.23,0.00),v60,z0,tPen\WObj:=wPaper;
    MoveL Offs(pOrigin,156.09,111.58,0.00),v40,fine,tPen\WObj:=wPaper;
    MoveL Offs(pOrigin,156.09,111.58,6.00),v60,z5,tPen\WObj:=wPaper;
    MoveL Offs(pOrigin,155.72,114.83,6.00),vTravel,z5,tPen\WObj:=wPaper;
    MoveL Offs(pOrigin,155.72,114.83,0.00),v60,z0,tPen\WObj:=wPaper;
    MoveL Offs(pOrigin,149.71,120.84,0.00),v40,fine,tPen\WObj:=wPaper;
    MoveL Offs(pOrigin,149.71,120.84,6.00),v60,z5,tPen\WObj:=wPaper;
    MoveL Offs(pOrigin,152.56,120.98,6.00),vTravel,z5,tPen\WObj:=wPaper;
    MoveL Offs(pOrigin,152.56,120.98,0.00),v60,z0,tPen\WObj:=wPaper;
    MoveL Offs(pOrigin,166.38,107.16,0.00),v40,z0,tPen\WObj:=wPaper;
    MoveL Offs(pOrigin,167.13,107.91,0.00),v40,z0,tPen\WObj:=wPaper;
    MoveL Offs(pOrigin,157.51,117.52,0.00),v40,z0,tPen\WObj:=wPaper;
    MoveL Offs(pOrigin,157.31,117.28,0.00),v40,z0,tPen\WObj:=wPaper;
    MoveL Offs(pOrigin,155.66,115.63,0.00),v40,z0,tPen\WObj:=wPaper;
    MoveL Offs(pOrigin,156.70,115.18,0.00),v40,z0,tPen\WObj:=wPaper;
    MoveL Offs(pOrigin,158.51,116.98,0.00),v40,z0,tPen\WObj:=wPaper;
    MoveL Offs(pOrigin,157.99,116.38,0.00),v40,z0,tPen\WObj:=wPaper;
    MoveL Offs(pOrigin,150.34,116.38,0.00),v40,z0,tPen\WObj:=wPaper;
    MoveL Offs(pOrigin,149.81,115.76,0.00),v40,z0,tPen\WObj:=wPaper;
    MoveL Offs(pOrigin,151.77,117.71,0.00),v40,fine,tPen\WObj:=wPaper;
    MoveL Offs(pOrigin,151.77,117.71,6.00),v60,z5,tPen\WObj:=wPaper;
    MoveL Offs(pOrigin,149.97,117.41,6.00),vTravel,z5,tPen\WObj:=wPaper;
    MoveL Offs(pOrigin,149.97,117.41,0.00),v60,z0,tPen\WObj:=wPaper;
    MoveL Offs(pOrigin,148.17,115.60,0.00),v40,z0,tPen\WObj:=wPaper;
    MoveL Offs(pOrigin,148.23,114.86,0.00),v40,z0,tPen\WObj:=wPaper;
    MoveL Offs(pOrigin,143.73,119.36,0.00),v40,z0,tPen\WObj:=wPaper;
    MoveL Offs(pOrigin,144.13,119.04,0.00),v40,z0,tPen\WObj:=wPaper;
    MoveL Offs(pOrigin,142.93,117.84,0.00),v40,fine,tPen\WObj:=wPaper;
    MoveL Offs(pOrigin,142.93,117.84,6.00),v60,z5,tPen\WObj:=wPaper;
    MoveL Offs(pOrigin,144.19,115.92,6.00),vTravel,z5,tPen\WObj:=wPaper;
    MoveL Offs(pOrigin,144.19,115.92,0.00),v60,z0,tPen\WObj:=wPaper;
    MoveL Offs(pOrigin,145.69,114.41,0.00),v40,fine,tPen\WObj:=wPaper;
    MoveL Offs(pOrigin,145.69,114.41,6.00),v60,z5,tPen\WObj:=wPaper;
    MoveL Offs(pOrigin,146.89,114.71,6.00),vTravel,z5,tPen\WObj:=wPaper;
    MoveL Offs(pOrigin,146.89,114.71,0.00),v60,z0,tPen\WObj:=wPaper;
    MoveL Offs(pOrigin,145.23,116.36,0.00),v40,fine,tPen\WObj:=wPaper;
    MoveL Offs(pOrigin,145.23,116.36,6.00),v60,z5,tPen\WObj:=wPaper;
    MoveL Offs(pOrigin,146.67,115.60,6.00),vTravel,z5,tPen\WObj:=wPaper;
    MoveL Offs(pOrigin,146.67,115.60,0.00),v60,z0,tPen\WObj:=wPaper;
    MoveL Offs(pOrigin,148.17,117.10,0.00),v40,fine,tPen\WObj:=wPaper;
    MoveL Offs(pOrigin,148.17,117.10,6.00),v60,z5,tPen\WObj:=wPaper;
    MoveL Offs(pOrigin,147.36,115.93,6.00),vTravel,z5,tPen\WObj:=wPaper;
    MoveL Offs(pOrigin,147.36,115.93,0.00),v60,z0,tPen\WObj:=wPaper;
    MoveL Offs(pOrigin,143.54,114.86,0.00),v40,fine,tPen\WObj:=wPaper;
    MoveL Offs(pOrigin,143.54,114.86,6.00),v60,z5,tPen\WObj:=wPaper;
    MoveL Offs(pOrigin,143.74,113.37,6.00),vTravel,z5,tPen\WObj:=wPaper;
    MoveL Offs(pOrigin,143.74,113.37,0.00),v60,z0,tPen\WObj:=wPaper;
    MoveL Offs(pOrigin,146.75,110.37,0.00),v40,z0,tPen\WObj:=wPaper;
    MoveL Offs(pOrigin,146.65,111.11,0.00),v40,z0,tPen\WObj:=wPaper;
    MoveL Offs(pOrigin,148.16,112.61,0.00),v40,fine,tPen\WObj:=wPaper;
    MoveL Offs(pOrigin,148.16,112.61,6.00),v60,z5,tPen\WObj:=wPaper;
    MoveL Offs(pOrigin,149.58,115.00,6.00),vTravel,z5,tPen\WObj:=wPaper;
    MoveL Offs(pOrigin,149.58,115.00,0.00),v60,z0,tPen\WObj:=wPaper;
    MoveL Offs(pOrigin,144.77,119.81,0.00),v40,fine,tPen\WObj:=wPaper;
    MoveL Offs(pOrigin,144.77,119.81,6.00),v60,z5,tPen\WObj:=wPaper;
    MoveL Offs(pOrigin,143.96,112.90,6.00),vTravel,z5,tPen\WObj:=wPaper;
    MoveL Offs(pOrigin,143.96,112.90,0.00),v60,z0,tPen\WObj:=wPaper;
    MoveL Offs(pOrigin,142.46,111.39,0.00),v40,fine,tPen\WObj:=wPaper;
    MoveL Offs(pOrigin,142.46,111.39,6.00),v60,z5,tPen\WObj:=wPaper;
    MoveL Offs(pOrigin,139.71,112.31,6.00),vTravel,z5,tPen\WObj:=wPaper;
    MoveL Offs(pOrigin,139.71,112.31,0.00),v60,z0,tPen\WObj:=wPaper;
    MoveL Offs(pOrigin,133.98,112.31,0.00),v40,z0,tPen\WObj:=wPaper;
    MoveL Offs(pOrigin,123.99,111.04,0.00),v40,fine,tPen\WObj:=wPaper;
    MoveL Offs(pOrigin,123.99,111.04,6.00),v60,z5,tPen\WObj:=wPaper;
    MoveL Offs(pOrigin,123.67,112.53,6.00),vTravel,z5,tPen\WObj:=wPaper;
    MoveL Offs(pOrigin,123.67,112.53,0.00),v60,z0,tPen\WObj:=wPaper;
    MoveL Offs(pOrigin,122.02,114.19,0.00),v40,z0,tPen\WObj:=wPaper;
  ENDPROC

